LIN {X 0,Y 525.321,Z 367.806,A -85,B 0,C 180,E1 -4749.038,E2 -4749.038} C_VEL
LIN {X 0,Y 524.882,Z 392.684,A -85,B 0,C 180,E1 -4751.929,E2 -4751.929} C_VEL
LIN {X 0,Y 524.49,Z 417.897,A -85,B 0,C 180,E1 -4754.808,E2 -4754.808} C_VEL
LIN {X 0,Y 525.888,Z 431.517,A -85,B 0,C 180,E1 -4755.052,E2 -4755.052} C_VEL
LIN {X 0,Y 525.465,Z 528.308,A -85,B 0,C 180,E1 -4756.39,E2 -4756.39} C_VEL
LIN {X 0,Y 525.226,Z 541.664,A -85,B 0,C 180,E1 -4756.729,E2 -4756.729} C_VEL
LIN {X 0,Y 524.966,Z 553.932,A -85,B 0,C 180,E1 -4757.19,E2 -4757.19} C_VEL
LIN {X 0,Y 524.718,Z 566.459,A -85,B 0,C 180,E1 -4757.828,E2 -4757.828} C_VEL
LIN {X 0,Y 524.441,Z 578.107,A -85,B 0,C 180,E1 -4758.6,E2 -4758.6} C_VEL
LIN {X 0,Y 524.161,Z 588.71,A -85,B 0,C 180,E1 -4759.474,E2 -4759.474} C_VEL
LIN {X 0,Y 523.963,Z 597.402,A -85,B 0,C 180,E1 -4760.348,E2 -4760.348} C_VEL
LIN {X 0,Y 523.771,Z 605.435,A -85,B 0,C 180,E1 -4761.318,E2 -4761.318} C_VEL
LIN {X 0,Y 523.629,Z 613.302,A -85,B 0,C 180,E1 -4762.481,E2 -4762.481} C_VEL
LIN {X 0,Y 523.502,Z 620.559,A -85,B 0,C 180,E1 -4763.835,E2 -4763.835} C_VEL
LIN {X 0,Y 523.411,Z 625.392,A -85,B 0,C 180,E1 -4764.993,E2 -4764.993} C_VEL
LIN {X 0,Y 523.475,Z 629.106,A -85,B 0,C 180,E1 -4766.151,E2 -4766.151} C_VEL
LIN {X 0,Y 523.397,Z 631.008,A -85,B 0,C 180,E1 -4766.921,E2 -4766.921} C_VEL
LIN {X 0,Y 523.345,Z 632.435,A -85,B 0,C 180,E1 -4767.691,E2 -4767.691} C_VEL
LIN {X 0,Y 523.279,Z 634.074,A -85,B 0,C 180,E1 -4769.23,E2 -4769.23} C_VEL
LIN {X 0,Y 523.278,Z 634.296,A -85,B 0,C 180,E1 -4770,E2 -4770} C_VEL
LIN {X 0,Y 523.279,Z 634.074,A -85,B 0,C 180,E1 -4770.77,E2 -4770.77} C_VEL
LIN {X 0,Y 523.345,Z 632.438,A -85,B 0,C 180,E1 -4772.309,E2 -4772.309} C_VEL
LIN {X 0,Y 523.397,Z 631.011,A -85,B 0,C 180,E1 -4773.079,E2 -4773.079} C_VEL
LIN {X 0,Y 523.441,Z 628.004,A -85,B 0,C 180,E1 -4774.235,E2 -4774.235} C_VEL
LIN {X 0,Y 523.464,Z 623.93,A -85,B 0,C 180,E1 -4775.393,E2 -4775.393} C_VEL
LIN {X 0,Y 523.516,Z 618.58,A -85,B 0,C 180,E1 -4776.574,E2 -4776.574} C_VEL
LIN {X 0,Y 523.649,Z 612.112,A -85,B 0,C 180,E1 -4777.713,E2 -4777.713} C_VEL
LIN {X 0,Y 523.821,Z 603.92,A -85,B 0,C 180,E1 -4778.876,E2 -4778.876} C_VEL
LIN {X 0,Y 524.017,Z 595.588,A -85,B 0,C 180,E1 -4779.846,E2 -4779.846} C_VEL
LIN {X 0,Y 524.277,Z 585.449,A -85,B 0,C 180,E1 -4780.817,E2 -4780.817} C_VEL
LIN {X 0,Y 524.576,Z 573.997,A -85,B 0,C 180,E1 -4781.693,E2 -4781.693} C_VEL
LIN {X 0,Y 524.816,Z 562.855,A -85,B 0,C 180,E1 -4782.372,E2 -4782.372} C_VEL
LIN {X 0,Y 525.058,Z 550.507,A -85,B 0,C 180,E1 -4782.956,E2 -4782.956} C_VEL
LIN {X 0,Y 525.318,Z 537.59,A -85,B 0,C 180,E1 -4783.392,E2 -4783.392} C_VEL
LIN {X 0,Y 525.501,Z 523.939,A -85,B 0,C 180,E1 -4783.683,E2 -4783.683} C_VEL
LIN {X 0,Y 525.776,Z 428.93,A -85,B 0,C 180,E1 -4784.986,E2 -4784.986} C_VEL
LIN {X 0,Y 524.48,Z 417.737,A -85,B 0,C 180,E1 -4785.202,E2 -4785.202} C_VEL
LIN {X 0,Y 524.855,Z 393.85,A -85,B 0,C 180,E1 -4787.937,E2 -4787.937} C_VEL
LIN {X 0,Y 525.421,Z 366.009,A -85,B 0,C 180,E1 -4791.17,E2 -4791.17} C_VEL
LIN {X 0,Y 525.911,Z 339.704,A -85,B 0,C 180,E1 -4794.263,E2 -4794.263} C_VEL
LIN {X 0,Y 526.305,Z 318.022,A -85,B 0,C 180,E1 -4796.856,E2 -4796.856} C_VEL
LIN {X 0,Y 523.957,Z 306.361,A -85,B 0,C 180,E1 -4798.421,E2 -4798.421} C_VEL
LIN {X 0,Y 523.907,Z 306.224,A -85,B 0,C 180,E1 -4801.544,E2 -4801.544} C_VEL
LIN {X 0,Y 523.909,Z 306.226,A -85,B 0,C 180,E1 -4804.291,E2 -4804.291} C_VEL
LIN {X 0,Y 523.878,Z 306.229,A -85,B 0,C 180,E1 -4807.673,E2 -4807.673} C_VEL
LIN {X 0,Y 523.909,Z 306.223,A -85,B 0,C 180,E1 -4810.126,E2 -4810.126} C_VEL
LIN {X 0,Y 523.875,Z 306.224,A -85,B 0,C 180,E1 -4813.171,E2 -4813.171} C_VEL
LIN {X 0,Y 523.919,Z 306.214,A -85,B 0,C 180,E1 -4815.77,E2 -4815.77} C_VEL
LIN {X 0,Y 523.89,Z 306.223,A -85,B 0,C 180,E1 -4818.903,E2 -4818.903} C_VEL
LIN {X 0,Y 523.895,Z 306.213,A -85,B 0,C 180,E1 -4821.896,E2 -4821.896} C_VEL
LIN {X 0,Y 523.907,Z 306.212,A -85,B 0,C 180,E1 -4824.912,E2 -4824.912} C_VEL
LIN {X 0,Y 523.928,Z 306.222,A -85,B 0,C 180,E1 -4827.679,E2 -4827.679} C_VEL
LIN {X 0,Y 523.946,Z 306.211,A -85,B 0,C 180,E1 -4830.676,E2 -4830.676} C_VEL
LIN {X 0,Y 523.894,Z 306.226,A -85,B 0,C 180,E1 -4833.724,E2 -4833.724} C_VEL
LIN {X 0,Y 523.901,Z 306.222,A -85,B 0,C 180,E1 -4836.269,E2 -4836.269} C_VEL
LIN {X 0,Y 523.937,Z 306.208,A -85,B 0,C 180,E1 -4838.766,E2 -4838.766} C_VEL
LIN {X 0,Y 523.928,Z 306.214,A -85,B 0,C 180,E1 -4841.22,E2 -4841.22} C_VEL
LIN {X 0,Y 523.912,Z 306.226,A -85,B 0,C 180,E1 -4843.638,E2 -4843.638} C_VEL
LIN {X 0,Y 523.921,Z 306.219,A -85,B 0,C 180,E1 -4846.027,E2 -4846.027} C_VEL
LIN {X 0,Y 523.98,Z 306.211,A -85,B 0,C 180,E1 -4849.177,E2 -4849.177} C_VEL
LIN {X 0,Y 523.988,Z 306.209,A -85,B 0,C 180,E1 -4852.292,E2 -4852.292} C_VEL
LIN {X 0,Y 524.057,Z 306.198,A -85,B 0,C 180,E1 -4854.613,E2 -4854.613} C_VEL
LIN {X 0,Y 524.092,Z 306.206,A -85,B 0,C 180,E1 -4857.694,E2 -4857.694} C_VEL
LIN {X 0,Y 524.083,Z 306.197,A -85,B 0,C 180,E1 -4860,E2 -4860} C_VEL
LIN {X 0,Y 524.025,Z 306.205,A -85,B 0,C 180,E1 -4863.075,E2 -4863.075} C_VEL
LIN {X 0,Y 523.999,Z 306.208,A -85,B 0,C 180,E1 -4866.16,E2 -4866.16} C_VEL
LIN {X 0,Y 523.97,Z 306.212,A -85,B 0,C 180,E1 -4869.262,E2 -4869.262} C_VEL
LIN {X 0,Y 523.988,Z 306.216,A -85,B 0,C 180,E1 -4871.736,E2 -4871.736} C_VEL
LIN {X 0,Y 523.975,Z 306.208,A -85,B 0,C 180,E1 -4875.048,E2 -4875.048} C_VEL
LIN {X 0,Y 523.907,Z 306.223,A -85,B 0,C 180,E1 -4877.971,E2 -4877.971} C_VEL
LIN {X 0,Y 523.944,Z 306.212,A -85,B 0,C 180,E1 -4880.411,E2 -4880.411} C_VEL
LIN {X 0,Y 523.898,Z 306.221,A -85,B 0,C 180,E1 -4882.894,E2 -4882.894} C_VEL
LIN {X 0,Y 523.892,Z 306.229,A -85,B 0,C 180,E1 -4885.422,E2 -4885.422} C_VEL
LIN {X 0,Y 523.898,Z 306.213,A -85,B 0,C 180,E1 -4888.003,E2 -4888.003} C_VEL
LIN {X 0,Y 523.925,Z 306.208,A -85,B 0,C 180,E1 -4890.853,E2 -4890.853} C_VEL
LIN {X 0,Y 523.919,Z 306.224,A -85,B 0,C 180,E1 -4893.729,E2 -4893.729} C_VEL
LIN {X 0,Y 523.891,Z 306.22,A -85,B 0,C 180,E1 -4896.401,E2 -4896.401} C_VEL
LIN {X 0,Y 523.903,Z 306.216,A -85,B 0,C 180,E1 -4899.087,E2 -4899.087} C_VEL
LIN {X 0,Y 523.888,Z 306.223,A -85,B 0,C 180,E1 -4902.126,E2 -4902.126} C_VEL
LIN {X 0,Y 523.928,Z 306.223,A -85,B 0,C 180,E1 -4905.312,E2 -4905.312} C_VEL
LIN {X 0,Y 523.874,Z 306.219,A -85,B 0,C 180,E1 -4906.87,E2 -4906.87} C_VEL
LIN {X 0,Y 523.187,Z 306.312,A -85,B 0,C 180,E1 -4907.512,E2 -4907.512} C_VEL
LIN {X 0,Y 520.324,Z 306.668,A -85,B 0,C 180,E1 -4908.553,E2 -4908.553} C_VEL
LIN {X 0,Y 517.93,Z 306.972,A -85,B 0,C 180,E1 -4909.392,E2 -4909.392} C_VEL
LIN {X 0,Y 516.924,Z 307.092,A -85,B 0,C 180,E1 -4910.04,E2 -4910.04} C_VEL
LIN {X 0,Y 516.853,Z 307.099,A -85,B 0,C 180,E1 -4910.259,E2 -4910.259} C_VEL
LIN {X 0,Y 516.843,Z 307.102,A -85,B 0,C 180,E1 -4913.349,E2 -4913.349} C_VEL
LIN {X 0,Y 516.876,Z 307.096,A -85,B 0,C 180,E1 -4916.119,E2 -4916.119} C_VEL
LIN {X 0,Y 516.848,Z 307.102,A -85,B 0,C 180,E1 -4918.944,E2 -4918.944} C_VEL
LIN {X 0,Y 516.843,Z 307.094,A -85,B 0,C 180,E1 -4921.581,E2 -4921.581} C_VEL
LIN {X 0,Y 516.842,Z 307.1,A -85,B 0,C 180,E1 -4924.207,E2 -4924.207} C_VEL
LIN {X 0,Y 516.855,Z 307.102,A -85,B 0,C 180,E1 -4926.776,E2 -4926.776} C_VEL
LIN {X 0,Y 516.931,Z 307.093,A -85,B 0,C 180,E1 -4929.735,E2 -4929.735} C_VEL
LIN {X 0,Y 516.884,Z 307.07,A -85,B 0,C 180,E1 -4932.595,E2 -4932.595} C_VEL
LIN {X 0,Y 516.96,Z 307.275,A -85,B 0,C 180,E1 -4934.94,E2 -4934.94} C_VEL
LIN {X 0,Y 517.203,Z 308.319,A -85,B 0,C 180,E1 -4935.069,E2 -4935.069} C_VEL
LIN {X 0,Y 519.147,Z 313.948,A -85,B 0,C 180,E1 -4935.221,E2 -4935.221} C_VEL
LIN {X 0,Y 518.857,Z 387.345,A -85,B 0,C 180,E1 -4936.263,E2 -4936.263} C_VEL
LIN {X 0,Y 518.772,Z 400.457,A -85,B 0,C 180,E1 -4936.61,E2 -4936.61} C_VEL
LIN {X 0,Y 518.62,Z 413.364,A -85,B 0,C 180,E1 -4937.12,E2 -4937.12} C_VEL
LIN {X 0,Y 518.424,Z 425.059,A -85,B 0,C 180,E1 -4937.752,E2 -4937.752} C_VEL
LIN {X 0,Y 518.072,Z 436.629,A -85,B 0,C 180,E1 -4938.557,E2 -4938.557} C_VEL
LIN {X 0,Y 517.797,Z 446.757,A -85,B 0,C 180,E1 -4939.442,E2 -4939.442} C_VEL
LIN {X 0,Y 517.518,Z 455.832,A -85,B 0,C 180,E1 -4940.424,E2 -4940.424} C_VEL
LIN {X 0,Y 517.235,Z 464.615,A -85,B 0,C 180,E1 -4941.601,E2 -4941.601} C_VEL
LIN {X 0,Y 517.056,Z 470.802,A -85,B 0,C 180,E1 -4942.62,E2 -4942.62} C_VEL
LIN {X 0,Y 516.937,Z 476.425,A -85,B 0,C 180,E1 -4943.756,E2 -4943.756} C_VEL
LIN {X 0,Y 516.696,Z 481.059,A -85,B 0,C 180,E1 -4944.928,E2 -4944.928} C_VEL
LIN {X 0,Y 516.648,Z 484.586,A -85,B 0,C 180,E1 -4946.1,E2 -4946.1} C_VEL
LIN {X 0,Y 516.587,Z 486.413,A -85,B 0,C 180,E1 -4946.881,E2 -4946.881} C_VEL
LIN {X 0,Y 516.579,Z 487.788,A -85,B 0,C 180,E1 -4947.661,E2 -4947.661} C_VEL
LIN {X 0,Y 516.546,Z 489.367,A -85,B 0,C 180,E1 -4949.22,E2 -4949.22} C_VEL
LIN {X 0,Y 516.535,Z 489.601,A -85,B 0,C 180,E1 -4950,E2 -4950} C_VEL
LIN {X 0,Y 516.546,Z 489.421,A -85,B 0,C 180,E1 -4950.78,E2 -4950.78} C_VEL
LIN {X 0,Y 516.578,Z 487.91,A -85,B 0,C 180,E1 -4952.339,E2 -4952.339} C_VEL
LIN {X 0,Y 516.584,Z 486.591,A -85,B 0,C 180,E1 -4953.119,E2 -4953.119} C_VEL
LIN {X 0,Y 516.707,Z 483.784,A -85,B 0,C 180,E1 -4954.29,E2 -4954.29} C_VEL
LIN {X 0,Y 516.823,Z 479.981,A -85,B 0,C 180,E1 -4955.462,E2 -4955.462} C_VEL
LIN {X 0,Y 516.897,Z 474.869,A -85,B 0,C 180,E1 -4956.683,E2 -4956.683} C_VEL
LIN {X 0,Y 517.15,Z 467.686,A -85,B 0,C 180,E1 -4958.007,E2 -4958.007} C_VEL
LIN {X 0,Y 517.415,Z 459.672,A -85,B 0,C 180,E1 -4959.183,E2 -4959.183} C_VEL
LIN {X 0,Y 517.669,Z 451.454,A -85,B 0,C 180,E1 -4960.165,E2 -4960.165} C_VEL
LIN {X 0,Y 517.944,Z 442.436,A -85,B 0,C 180,E1 -4961.05,E2 -4961.05} C_VEL
LIN {X 0,Y 518.281,Z 431.958,A -85,B 0,C 180,E1 -4961.88,E2 -4961.88} C_VEL
LIN {X 0,Y 518.473,Z 420.319,A -85,B 0,C 180,E1 -4962.615,E2 -4962.615} C_VEL
LIN {X 0,Y 518.647,Z 408.922,A -85,B 0,C 180,E1 -4963.168,E2 -4963.168} C_VEL
LIN {X 0,Y 518.815,Z 396.128,A -85,B 0,C 180,E1 -4963.613,E2 -4963.613} C_VEL
LIN {X 0,Y 518.834,Z 383.996,A -85,B 0,C 180,E1 -4963.887,E2 -4963.887} C_VEL
LIN {X 0,Y 519.053,Z 313.676,A -85,B 0,C 180,E1 -4964.876,E2 -4964.876} C_VEL
LIN {X 0,Y 517.038,Z 307.902,A -85,B 0,C 180,E1 -4965.051,E2 -4965.051} C_VEL
LIN {X 0,Y 516.904,Z 307.157,A -85,B 0,C 180,E1 -4965.21,E2 -4965.21} C_VEL
LIN {X 0,Y 516.871,Z 307.068,A -85,B 0,C 180,E1 -4968.224,E2 -4968.224} C_VEL
LIN {X 0,Y 516.887,Z 307.104,A -85,B 0,C 180,E1 -4970.702,E2 -4970.702} C_VEL
LIN {X 0,Y 516.855,Z 307.102,A -85,B 0,C 180,E1 -4973.224,E2 -4973.224} C_VEL
LIN {X 0,Y 516.855,Z 307.099,A -85,B 0,C 180,E1 -4976.175,E2 -4976.175} C_VEL
LIN {X 0,Y 516.897,Z 307.095,A -85,B 0,C 180,E1 -4979.305,E2 -4979.305} C_VEL
LIN {X 0,Y 516.862,Z 307.101,A -85,B 0,C 180,E1 -4982.537,E2 -4982.537} C_VEL
LIN {X 0,Y 516.851,Z 307.1,A -85,B 0,C 180,E1 -4985.327,E2 -4985.327} C_VEL
LIN {X 0,Y 516.867,Z 307.102,A -85,B 0,C 180,E1 -4988.716,E2 -4988.716} C_VEL
LIN {X 0,Y 516.84,Z 307.098,A -85,B 0,C 180,E1 -4991.781,E2 -4991.781} C_VEL
LIN {X 0,Y 516.892,Z 307.098,A -85,B 0,C 180,E1 -4995.006,E2 -4995.006} C_VEL
LIN {X 0,Y 516.843,Z 307.106,A -85,B 0,C 180,E1 -4998.406,E2 -4998.406} C_VEL
LIN {X 0,Y 516.865,Z 307.089,A -85,B 0,C 180,E1 -5001.282,E2 -5001.282} C_VEL
LIN {X 0,Y 516.85,Z 307.101,A -85,B 0,C 180,E1 -5004.218,E2 -5004.218} C_VEL
LIN {X 0,Y 516.873,Z 307.096,A -85,B 0,C 180,E1 -5007.051,E2 -5007.051} C_VEL
LIN {X 0,Y 516.839,Z 307.089,A -85,B 0,C 180,E1 -5009.793,E2 -5009.793} C_VEL
LIN {X 0,Y 516.867,Z 307.094,A -85,B 0,C 180,E1 -5012.464,E2 -5012.464} C_VEL
LIN {X 0,Y 516.837,Z 307.103,A -85,B 0,C 180,E1 -5015.068,E2 -5015.068} C_VEL
LIN {X 0,Y 516.862,Z 307.096,A -85,B 0,C 180,E1 -5017.621,E2 -5017.621} C_VEL
LIN {X 0,Y 516.906,Z 307.092,A -85,B 0,C 180,E1 -5020.129,E2 -5020.129} C_VEL
LIN {X 0,Y 516.863,Z 307.096,A -85,B 0,C 180,E1 -5023.408,E2 -5023.408} C_VEL
LIN {X 0,Y 516.857,Z 307.094,A -85,B 0,C 180,E1 -5025.832,E2 -5025.832} C_VEL
LIN {X 0,Y 516.933,Z 307.09,A -85,B 0,C 180,E1 -5029.027,E2 -5029.027} C_VEL
LIN {X 0,Y 516.916,Z 307.093,A -85,B 0,C 180,E1 -5032.186,E2 -5032.186} C_VEL
LIN {X 0,Y 516.97,Z 307.091,A -85,B 0,C 180,E1 -5034.539,E2 -5034.539} C_VEL
LIN {X 0,Y 517.063,Z 307.072,A -85,B 0,C 180,E1 -5037.663,E2 -5037.663} C_VEL
LIN {X 0,Y 517.08,Z 307.072,A -85,B 0,C 180,E1 -5040.779,E2 -5040.779} C_VEL
LIN {X 0,Y 516.935,Z 307.088,A -85,B 0,C 180,E1 -5043.117,E2 -5043.117} C_VEL
LIN {X 0,Y 516.974,Z 307.086,A -85,B 0,C 180,E1 -5046.244,E2 -5046.244} C_VEL
LIN {X 0,Y 516.921,Z 307.09,A -85,B 0,C 180,E1 -5049.39,E2 -5049.39} C_VEL
LIN {X 0,Y 516.897,Z 307.094,A -85,B 0,C 180,E1 -5052.565,E2 -5052.565} C_VEL
LIN {X 0,Y 516.936,Z 307.088,A -85,B 0,C 180,E1 -5055.146,E2 -5055.146} C_VEL
LIN {X 0,Y 516.869,Z 307.101,A -85,B 0,C 180,E1 -5058.224,E2 -5058.224} C_VEL
LIN {X 0,Y 516.897,Z 307.088,A -85,B 0,C 180,E1 -5060.702,E2 -5060.702} C_VEL
LIN {X 0,Y 516.877,Z 307.102,A -85,B 0,C 180,E1 -5064.074,E2 -5064.074} C_VEL
LIN {X 0,Y 516.836,Z 307.1,A -85,B 0,C 180,E1 -5066.663,E2 -5066.663} C_VEL
LIN {X 0,Y 516.902,Z 307.09,A -85,B 0,C 180,E1 -5069.524,E2 -5069.524} C_VEL
LIN {X 0,Y 516.888,Z 307.097,A -85,B 0,C 180,E1 -5072.543,E2 -5072.543} C_VEL
LIN {X 0,Y 516.844,Z 307.097,A -85,B 0,C 180,E1 -5075.327,E2 -5075.327} C_VEL
LIN {X 0,Y 516.867,Z 307.095,A -85,B 0,C 180,E1 -5078.717,E2 -5078.717} C_VEL
LIN {X 0,Y 516.877,Z 307.101,A -85,B 0,C 180,E1 -5081.779,E2 -5081.779} C_VEL
LIN {X 0,Y 516.892,Z 307.082,A -85,B 0,C 180,E1 -5085.008,E2 -5085.008} C_VEL
LIN {X 0,Y 516.848,Z 307.102,A -85,B 0,C 180,E1 -5088.407,E2 -5088.407} C_VEL
LIN {X 0,Y 516.87,Z 307.095,A -85,B 0,C 180,E1 -5091.284,E2 -5091.284} C_VEL
LIN {X 0,Y 516.847,Z 307.101,A -85,B 0,C 180,E1 -5094.674,E2 -5094.674} C_VEL
LIN {X 0,Y 516.888,Z 307.094,A -85,B 0,C 180,E1 -5097.458,E2 -5097.458} C_VEL
LIN {X 0,Y 516.901,Z 307.077,A -85,B 0,C 180,E1 -5100.695,E2 -5100.695} C_VEL
LIN {X 0,Y 516.935,Z 307.345,A -85,B 0,C 180,E1 -5101.406,E2 -5101.406} C_VEL
LIN {X 0,Y 519.378,Z 319.028,A -85,B 0,C 180,E1 -5102.987,E2 -5102.987} C_VEL
LIN {X 0,Y 519.069,Z 337.058,A -85,B 0,C 180,E1 -5105.183,E2 -5105.183} C_VEL
LIN {X 0,Y 518.527,Z 361.62,A -85,B 0,C 180,E1 -5108.116,E2 -5108.116} C_VEL
LIN {X 0,Y 518.001,Z 386.005,A -85,B 0,C 180,E1 -5110.997,E2 -5110.997} C_VEL
LIN {X 0,Y 517.539,Z 410.213,A -85,B 0,C 180,E1 -5113.837,E2 -5113.837} C_VEL
LIN {X 0,Y 517.48,Z 416.952,A -85,B 0,C 180,E1 -5114.6,E2 -5114.6} C_VEL
LIN {X 0,Y 519.009,Z 432.102,A -85,B 0,C 180,E1 -5114.872,E2 -5114.872} C_VEL
LIN {X 0,Y 518.531,Z 527.315,A -85,B 0,C 180,E1 -5116.205,E2 -5116.205} C_VEL
LIN {X 0,Y 518.275,Z 540.67,A -85,B 0,C 180,E1 -5116.547,E2 -5116.547} C_VEL
LIN {X 0,Y 518.014,Z 552.939,A -85,B 0,C 180,E1 -5117.015,E2 -5117.015} C_VEL
LIN {X 0,Y 517.708,Z 565.493,A -85,B 0,C 180,E1 -5117.663,E2 -5117.663} C_VEL
LIN {X 0,Y 517.439,Z 577.113,A -85,B 0,C 180,E1 -5118.443,E2 -5118.443} C_VEL
LIN {X 0,Y 517.134,Z 587.715,A -85,B 0,C 180,E1 -5119.329,E2 -5119.329} C_VEL
LIN {X 0,Y 516.911,Z 596.406,A -85,B 0,C 180,E1 -5120.215,E2 -5120.215} C_VEL
LIN {X 0,Y 516.711,Z 604.441,A -85,B 0,C 180,E1 -5121.198,E2 -5121.198} C_VEL
LIN {X 0,Y 516.554,Z 612.309,A -85,B 0,C 180,E1 -5122.377,E2 -5122.377} C_VEL
LIN {X 0,Y 516.435,Z 619.57,A -85,B 0,C 180,E1 -5123.75,E2 -5123.75} C_VEL
LIN {X 0,Y 516.382,Z 624.41,A -85,B 0,C 180,E1 -5124.925,E2 -5124.925} C_VEL
LIN {X 0,Y 516.43,Z 628.124,A -85,B 0,C 180,E1 -5126.098,E2 -5126.098} C_VEL
LIN {X 0,Y 516.352,Z 630.026,A -85,B 0,C 180,E1 -5126.879,E2 -5126.879} C_VEL
LIN {X 0,Y 516.304,Z 631.455,A -85,B 0,C 180,E1 -5127.66,E2 -5127.66} C_VEL
LIN {X 0,Y 516.265,Z 633.098,A -85,B 0,C 180,E1 -5129.22,E2 -5129.22} C_VEL
LIN {X 0,Y 516.261,Z 633.319,A -85,B 0,C 180,E1 -5130,E2 -5130} C_VEL
LIN {X 0,Y 516.265,Z 633.098,A -85,B 0,C 180,E1 -5130.78,E2 -5130.78} C_VEL
LIN {X 0,Y 516.304,Z 631.458,A -85,B 0,C 180,E1 -5132.34,E2 -5132.34} C_VEL
LIN {X 0,Y 516.352,Z 630.029,A -85,B 0,C 180,E1 -5133.121,E2 -5133.121} C_VEL
LIN {X 0,Y 516.387,Z 627.02,A -85,B 0,C 180,E1 -5134.293,E2 -5134.293} C_VEL
LIN {X 0,Y 516.404,Z 622.943,A -85,B 0,C 180,E1 -5135.467,E2 -5135.467} C_VEL
LIN {X 0,Y 516.489,Z 616.818,A -85,B 0,C 180,E1 -5136.812,E2 -5136.812} C_VEL
LIN {X 0,Y 516.585,Z 609.855,A -85,B 0,C 180,E1 -5138.016,E2 -5138.016} C_VEL
LIN {X 0,Y 516.769,Z 601.403,A -85,B 0,C 180,E1 -5139.195,E2 -5139.195} C_VEL
LIN {X 0,Y 517.006,Z 592.757,A -85,B 0,C 180,E1 -5140.178,E2 -5140.178} C_VEL
LIN {X 0,Y 517.318,Z 582.101,A -85,B 0,C 180,E1 -5141.162,E2 -5141.162} C_VEL
LIN {X 0,Y 517.578,Z 571.208,A -85,B 0,C 180,E1 -5141.976,E2 -5141.976} C_VEL
LIN {X 0,Y 517.86,Z 560.07,A -85,B 0,C 180,E1 -5142.64,E2 -5142.64} C_VEL
LIN {X 0,Y 518.18,Z 548.294,A -85,B 0,C 180,E1 -5143.181,E2 -5143.181} C_VEL
LIN {X 0,Y 518.403,Z 535.678,A -85,B 0,C 180,E1 -5143.599,E2 -5143.599} C_VEL
LIN {X 0,Y 518.601,Z 522.951,A -85,B 0,C 180,E1 -5143.868,E2 -5143.868} C_VEL
LIN {X 0,Y 518.903,Z 429.886,A -85,B 0,C 180,E1 -5145.162,E2 -5145.162} C_VEL
LIN {X 0,Y 517.455,Z 416.853,A -85,B 0,C 180,E1 -5145.406,E2 -5145.406} C_VEL
LIN {X 0,Y 517.899,Z 391.373,A -85,B 0,C 180,E1 -5148.37,E2 -5148.37} C_VEL
LIN {X 0,Y 518.44,Z 365.117,A -85,B 0,C 180,E1 -5151.47,E2 -5151.47} C_VEL
LIN {X 0,Y 518.976,Z 340.569,A -85,B 0,C 180,E1 -5154.395,E2 -5154.395} C_VEL
LIN {X 0,Y 519.465,Z 320.55,A -85,B 0,C 180,E1 -5156.819,E2 -5156.819} C_VEL
LIN {X 0,Y 518.03,Z 312.209,A -85,B 0,C 180,E1 -5157.917,E2 -5157.917} C_VEL
LIN {X 0,Y 516.899,Z 307.213,A -85,B 0,C 180,E1 -5158.638,E2 -5158.638} C_VEL
LIN {X 0,Y 516.877,Z 307.098,A -85,B 0,C 180,E1 -5161.11,E2 -5161.11} C_VEL
LIN {X 0,Y 516.879,Z 307.103,A -85,B 0,C 180,E1 -5163.961,E2 -5163.961} C_VEL
LIN {X 0,Y 516.812,Z 307.106,A -85,B 0,C 180,E1 -5166.751,E2 -5166.751} C_VEL
LIN {X 0,Y 516.854,Z 307.098,A -85,B 0,C 180,E1 -5169.723,E2 -5169.723} C_VEL
LIN {X 0,Y 516.837,Z 307.101,A -85,B 0,C 180,E1 -5172.835,E2 -5172.835} C_VEL
LIN {X 0,Y 516.891,Z 307.083,A -85,B 0,C 180,E1 -5175.006,E2 -5175.006} C_VEL
LIN {X 0,Y 516.88,Z 307.099,A -85,B 0,C 180,E1 -5178.402,E2 -5178.402} C_VEL
LIN {X 0,Y 516.867,Z 307.093,A -85,B 0,C 180,E1 -5181.283,E2 -5181.283} C_VEL
LIN {X 0,Y 516.844,Z 307.092,A -85,B 0,C 180,E1 -5184.672,E2 -5184.672} C_VEL
LIN {X 0,Y 516.887,Z 307.096,A -85,B 0,C 180,E1 -5187.457,E2 -5187.457} C_VEL
LIN {X 0,Y 516.914,Z 307.086,A -85,B 0,C 180,E1 -5190.695,E2 -5190.695} C_VEL
LIN {X 0,Y 516.873,Z 307.102,A -85,B 0,C 180,E1 -5193.818,E2 -5193.818} C_VEL
LIN {X 0,Y 516.85,Z 307.097,A -85,B 0,C 180,E1 -5196.775,E2 -5196.775} C_VEL
LIN {X 0,Y 516.929,Z 307.087,A -85,B 0,C 180,E1 -5199.732,E2 -5199.732} C_VEL
LIN {X 0,Y 516.886,Z 307.094,A -85,B 0,C 180,E1 -5202.595,E2 -5202.595} C_VEL
LIN {X 0,Y 516.934,Z 307.089,A -85,B 0,C 180,E1 -5205.03,E2 -5205.03} C_VEL
LIN {X 0,Y 516.958,Z 307.087,A -85,B 0,C 180,E1 -5208.233,E2 -5208.233} C_VEL
LIN {X 0,Y 516.92,Z 307.094,A -85,B 0,C 180,E1 -5211.399,E2 -5211.399} C_VEL
LIN {X 0,Y 516.976,Z 307.086,A -85,B 0,C 180,E1 -5213.756,E2 -5213.756} C_VEL
LIN {X 0,Y 516.937,Z 307.088,A -85,B 0,C 180,E1 -5216.883,E2 -5216.883} C_VEL
LIN {X 0,Y 517.08,Z 307.072,A -85,B 0,C 180,E1 -5219.221,E2 -5219.221} C_VEL
LIN {X 0,Y 517.064,Z 307.072,A -85,B 0,C 180,E1 -5222.337,E2 -5222.337} C_VEL
LIN {X 0,Y 516.964,Z 307.083,A -85,B 0,C 180,E1 -5226.244,E2 -5226.244} C_VEL
LIN {X 0,Y 516.927,Z 307.091,A -85,B 0,C 180,E1 -5229.39,E2 -5229.39} C_VEL
LIN {X 0,Y 516.944,Z 307.092,A -85,B 0,C 180,E1 -5231.807,E2 -5231.807} C_VEL
LIN {X 0,Y 516.928,Z 307.086,A -85,B 0,C 180,E1 -5235.143,E2 -5235.143} C_VEL
LIN {X 0,Y 516.869,Z 307.097,A -85,B 0,C 180,E1 -5238.224,E2 -5238.224} C_VEL
LIN {X 0,Y 516.894,Z 307.09,A -85,B 0,C 180,E1 -5240.702,E2 -5240.702} C_VEL
LIN {X 0,Y 516.848,Z 307.103,A -85,B 0,C 180,E1 -5243.225,E2 -5243.225} C_VEL
LIN {X 0,Y 516.873,Z 307.094,A -85,B 0,C 180,E1 -5246.182,E2 -5246.182} C_VEL
LIN {X 0,Y 516.896,Z 307.085,A -85,B 0,C 180,E1 -5249.306,E2 -5249.306} C_VEL
LIN {X 0,Y 516.887,Z 307.091,A -85,B 0,C 180,E1 -5252.543,E2 -5252.543} C_VEL
LIN {X 0,Y 516.854,Z 307.106,A -85,B 0,C 180,E1 -5255.329,E2 -5255.329} C_VEL
LIN {X 0,Y 516.87,Z 307.09,A -85,B 0,C 180,E1 -5257.943,E2 -5257.943} C_VEL
LIN {X 0,Y 516.842,Z 307.095,A -85,B 0,C 180,E1 -5260.746,E2 -5260.746} C_VEL
LIN {X 0,Y 516.876,Z 307.098,A -85,B 0,C 180,E1 -5263.904,E2 -5263.904} C_VEL
LIN {X 0,Y 516.825,Z 307.097,A -85,B 0,C 180,E1 -5266.872,E2 -5266.872} C_VEL
LIN {X 0,Y 516.855,Z 307.105,A -85,B 0,C 180,E1 -5269.594,E2 -5269.594} C_VEL
LIN {X 0,Y 516.853,Z 307.099,A -85,B 0,C 180,E1 -5270.259,E2 -5270.259} C_VEL
LIN {X 0,Y 516.215,Z 307.182,A -85,B 0,C 180,E1 -5270.909,E2 -5270.909} C_VEL
LIN {X 0,Y 513.368,Z 307.541,A -85,B 0,C 180,E1 -5271.965,E2 -5271.965} C_VEL
LIN {X 0,Y 510.938,Z 307.845,A -85,B 0,C 180,E1 -5272.815,E2 -5272.815} C_VEL
LIN {X 0,Y 509.887,Z 307.973,A -85,B 0,C 180,E1 -5273.471,E2 -5273.471} C_VEL
LIN {X 0,Y 509.799,Z 307.982,A -85,B 0,C 180,E1 -5273.694,E2 -5273.694} C_VEL
LIN {X 0,Y 509.831,Z 307.973,A -85,B 0,C 180,E1 -5276.538,E2 -5276.538} C_VEL
LIN {X 0,Y 509.804,Z 307.986,A -85,B 0,C 180,E1 -5279.332,E2 -5279.332} C_VEL
LIN {X 0,Y 509.826,Z 307.963,A -85,B 0,C 180,E1 -5282.051,E2 -5282.051} C_VEL
LIN {X 0,Y 509.783,Z 307.981,A -85,B 0,C 180,E1 -5284.699,E2 -5284.699} C_VEL
LIN {X 0,Y 509.825,Z 307.972,A -85,B 0,C 180,E1 -5287.459,E2 -5287.459} C_VEL
LIN {X 0,Y 509.907,Z 307.967,A -85,B 0,C 180,E1 -5289.845,E2 -5289.845} C_VEL
LIN {X 0,Y 509.82,Z 307.947,A -85,B 0,C 180,E1 -5293.173,E2 -5293.173} C_VEL
LIN {X 0,Y 509.902,Z 308.111,A -85,B 0,C 180,E1 -5294.711,E2 -5294.711} C_VEL
LIN {X 0,Y 510.083,Z 308.927,A -85,B 0,C 180,E1 -5294.84,E2 -5294.84} C_VEL
LIN {X 0,Y 512.276,Z 315.271,A -85,B 0,C 180,E1 -5295.022,E2 -5295.022} C_VEL
LIN {X 0,Y 512.032,Z 388.351,A -85,B 0,C 180,E1 -5296.077,E2 -5296.077} C_VEL
LIN {X 0,Y 511.929,Z 401.454,A -85,B 0,C 180,E1 -5296.428,E2 -5296.428} C_VEL
LIN {X 0,Y 511.766,Z 414.356,A -85,B 0,C 180,E1 -5296.944,E2 -5296.944} C_VEL
LIN {X 0,Y 511.589,Z 425.155,A -85,B 0,C 180,E1 -5297.529,E2 -5297.529} C_VEL
LIN {X 0,Y 511.227,Z 436.344,A -85,B 0,C 180,E1 -5298.301,E2 -5298.301} C_VEL
LIN {X 0,Y 510.917,Z 446.693,A -85,B 0,C 180,E1 -5299.198,E2 -5299.198} C_VEL
LIN {X 0,Y 510.663,Z 455.133,A -85,B 0,C 180,E1 -5300.094,E2 -5300.094} C_VEL
LIN {X 0,Y 510.345,Z 462.903,A -85,B 0,C 180,E1 -5301.088,E2 -5301.088} C_VEL
LIN {X 0,Y 510.122,Z 470.588,A -85,B 0,C 180,E1 -5302.3,E2 -5302.3} C_VEL
LIN {X 0,Y 509.954,Z 477.406,A -85,B 0,C 180,E1 -5303.67,E2 -5303.67} C_VEL
LIN {X 0,Y 509.699,Z 482.038,A -85,B 0,C 180,E1 -5304.858,E2 -5304.858} C_VEL
LIN {X 0,Y 509.633,Z 485.566,A -85,B 0,C 180,E1 -5306.046,E2 -5306.046} C_VEL
LIN {X 0,Y 509.565,Z 487.393,A -85,B 0,C 180,E1 -5306.838,E2 -5306.838} C_VEL
LIN {X 0,Y 509.568,Z 488.765,A -85,B 0,C 180,E1 -5307.629,E2 -5307.629} C_VEL
LIN {X 0,Y 509.533,Z 490.343,A -85,B 0,C 180,E1 -5309.21,E2 -5309.21} C_VEL
LIN {X 0,Y 509.521,Z 490.577,A -85,B 0,C 180,E1 -5310,E2 -5310} C_VEL
LIN {X 0,Y 509.533,Z 490.396,A -85,B 0,C 180,E1 -5310.79,E2 -5310.79} C_VEL
LIN {X 0,Y 509.568,Z 488.885,A -85,B 0,C 180,E1 -5312.371,E2 -5312.371} C_VEL
LIN {X 0,Y 509.562,Z 487.568,A -85,B 0,C 180,E1 -5313.163,E2 -5313.163} C_VEL
LIN {X 0,Y 509.695,Z 484.761,A -85,B 0,C 180,E1 -5314.349,E2 -5314.349} C_VEL
LIN {X 0,Y 509.84,Z 480.956,A -85,B 0,C 180,E1 -5315.537,E2 -5315.537} C_VEL
LIN {X 0,Y 509.916,Z 475.854,A -85,B 0,C 180,E1 -5316.773,E2 -5316.773} C_VEL
LIN {X 0,Y 510.194,Z 468.66,A -85,B 0,C 180,E1 -5318.117,E2 -5318.117} C_VEL
LIN {X 0,Y 510.484,Z 460.644,A -85,B 0,C 180,E1 -5319.309,E2 -5319.309} C_VEL
LIN {X 0,Y 510.753,Z 452.426,A -85,B 0,C 180,E1 -5320.304,E2 -5320.304} C_VEL
LIN {X 0,Y 511.046,Z 443.407,A -85,B 0,C 180,E1 -5321.201,E2 -5321.201} C_VEL
LIN {X 0,Y 511.412,Z 432.926,A -85,B 0,C 180,E1 -5322.042,E2 -5322.042} C_VEL
LIN {X 0,Y 511.617,Z 421.286,A -85,B 0,C 180,E1 -5322.787,E2 -5322.787} C_VEL
LIN {X 0,Y 511.795,Z 409.887,A -85,B 0,C 180,E1 -5323.348,E2 -5323.348} C_VEL
LIN {X 0,Y 511.971,Z 397.086,A -85,B 0,C 180,E1 -5323.799,E2 -5323.799} C_VEL
LIN {X 0,Y 511.993,Z 384.94,A -85,B 0,C 180,E1 -5324.076,E2 -5324.076} C_VEL
LIN {X 0,Y 512.276,Z 315.283,A -85,B 0,C 180,E1 -5325.068,E2 -5325.068} C_VEL
LIN {X 0,Y 510.03,Z 308.901,A -85,B 0,C 180,E1 -5325.254,E2 -5325.254} C_VEL
LIN {X 0,Y 509.838,Z 308.05,A -85,B 0,C 180,E1 -5325.415,E2 -5325.415} C_VEL
LIN {X 0,Y 509.828,Z 307.949,A -85,B 0,C 180,E1 -5328.485,E2 -5328.485} C_VEL
LIN {X 0,Y 509.834,Z 307.977,A -85,B 0,C 180,E1 -5331.002,E2 -5331.002} C_VEL
LIN {X 0,Y 509.811,Z 307.977,A -85,B 0,C 180,E1 -5333.564,E2 -5333.564} C_VEL
LIN {X 0,Y 509.796,Z 307.978,A -85,B 0,C 180,E1 -5336.351,E2 -5336.351} C_VEL
LIN {X 0,Y 509.83,Z 307.973,A -85,B 0,C 180,E1 -5338.847,E2 -5338.847} C_VEL
LIN {X 0,Y 509.786,Z 307.979,A -85,B 0,C 180,E1 -5341.592,E2 -5341.592} C_VEL
LIN {X 0,Y 509.827,Z 307.978,A -85,B 0,C 180,E1 -5344.415,E2 -5344.415} C_VEL
LIN {X 0,Y 509.789,Z 307.975,A -85,B 0,C 180,E1 -5347.342,E2 -5347.342} C_VEL
LIN {X 0,Y 509.809,Z 307.981,A -85,B 0,C 180,E1 -5350.384,E2 -5350.384} C_VEL
LIN {X 0,Y 509.788,Z 307.971,A -85,B 0,C 180,E1 -5353.574,E2 -5353.574} C_VEL
LIN {X 0,Y 509.786,Z 307.985,A -85,B 0,C 180,E1 -5356.424,E2 -5356.424} C_VEL
LIN {X 0,Y 509.807,Z 307.97,A -85,B 0,C 180,E1 -5359.614,E2 -5359.614} C_VEL
LIN {X 0,Y 509.798,Z 307.979,A -85,B 0,C 180,E1 -5362.657,E2 -5362.657} C_VEL
LIN {X 0,Y 509.832,Z 307.974,A -85,B 0,C 180,E1 -5365.8,E2 -5365.8} C_VEL
LIN {X 0,Y 509.831,Z 307.967,A -85,B 0,C 180,E1 -5368.721,E2 -5368.721} C_VEL
LIN {X 0,Y 509.808,Z 307.965,A -85,B 0,C 180,E1 -5371.916,E2 -5371.916} C_VEL
LIN {X 0,Y 509.794,Z 307.984,A -85,B 0,C 180,E1 -5374.699,E2 -5374.699} C_VEL
LIN {X 0,Y 509.816,Z 307.974,A -85,B 0,C 180,E1 -5377.459,E2 -5377.459} C_VEL
LIN {X 0,Y 509.881,Z 307.964,A -85,B 0,C 180,E1 -5379.843,E2 -5379.843} C_VEL
LIN {X 0,Y 509.81,Z 307.976,A -85,B 0,C 180,E1 -5383.172,E2 -5383.172} C_VEL
LIN {X 0,Y 509.832,Z 307.967,A -85,B 0,C 180,E1 -5385.633,E2 -5385.633} C_VEL
LIN {X 0,Y 509.898,Z 307.968,A -85,B 0,C 180,E1 -5388.874,E2 -5388.874} C_VEL
LIN {X 0,Y 509.868,Z 307.969,A -85,B 0,C 180,E1 -5392.077,E2 -5392.077} C_VEL
LIN {X 0,Y 509.923,Z 307.97,A -85,B 0,C 180,E1 -5394.464,E2 -5394.464} C_VEL
LIN {X 0,Y 510.034,Z 307.947,A -85,B 0,C 180,E1 -5397.631,E2 -5397.631} C_VEL
LIN {X 0,Y 510.029,Z 307.95,A -85,B 0,C 180,E1 -5400.79,E2 -5400.79} C_VEL
LIN {X 0,Y 509.879,Z 307.967,A -85,B 0,C 180,E1 -5403.161,E2 -5403.161} C_VEL
LIN {X 0,Y 509.928,Z 307.963,A -85,B 0,C 180,E1 -5406.33,E2 -5406.33} C_VEL
LIN {X 0,Y 509.873,Z 307.971,A -85,B 0,C 180,E1 -5408.721,E2 -5408.721} C_VEL
LIN {X 0,Y 509.892,Z 307.968,A -85,B 0,C 180,E1 -5411.932,E2 -5411.932} C_VEL
LIN {X 0,Y 509.887,Z 307.966,A -85,B 0,C 180,E1 -5415.242,E2 -5415.242} C_VEL
LIN {X 0,Y 509.829,Z 307.973,A -85,B 0,C 180,E1 -5418.485,E2 -5418.485} C_VEL
LIN {X 0,Y 509.838,Z 307.964,A -85,B 0,C 180,E1 -5421.002,E2 -5421.002} C_VEL
LIN {X 0,Y 509.811,Z 307.976,A -85,B 0,C 180,E1 -5423.564,E2 -5423.564} C_VEL
LIN {X 0,Y 509.81,Z 307.979,A -85,B 0,C 180,E1 -5426.357,E2 -5426.357} C_VEL
LIN {X 0,Y 509.842,Z 307.968,A -85,B 0,C 180,E1 -5428.846,E2 -5428.846} C_VEL
LIN {X 0,Y 509.812,Z 307.978,A -85,B 0,C 180,E1 -5431.591,E2 -5431.591} C_VEL
LIN {X 0,Y 509.827,Z 307.975,A -85,B 0,C 180,E1 -5434.415,E2 -5434.415} C_VEL
LIN {X 0,Y 509.774,Z 307.982,A -85,B 0,C 180,E1 -5437.345,E2 -5437.345} C_VEL
LIN {X 0,Y 509.808,Z 307.981,A -85,B 0,C 180,E1 -5440.385,E2 -5440.385} C_VEL
LIN {X 0,Y 509.79,Z 307.976,A -85,B 0,C 180,E1 -5443.059,E2 -5443.059} C_VEL
LIN {X 0,Y 509.802,Z 307.97,A -85,B 0,C 180,E1 -5445.796,E2 -5445.796} C_VEL
LIN {X 0,Y 509.801,Z 307.978,A -85,B 0,C 180,E1 -5448.57,E2 -5448.57} C_VEL
LIN {X 0,Y 509.812,Z 307.977,A -85,B 0,C 180,E1 -5451.659,E2 -5451.659} C_VEL
LIN {X 0,Y 509.805,Z 307.978,A -85,B 0,C 180,E1 -5454.621,E2 -5454.621} C_VEL
LIN {X 0,Y 509.854,Z 307.971,A -85,B 0,C 180,E1 -5457.481,E2 -5457.481} C_VEL
LIN {X 0,Y 509.865,Z 307.953,A -85,B 0,C 180,E1 -5460.93,E2 -5460.93} C_VEL
LIN {X 0,Y 509.878,Z 308.244,A -85,B 0,C 180,E1 -5461.203,E2 -5461.203} C_VEL
LIN {X 0,Y 512.493,Z 320.566,A -85,B 0,C 180,E1 -5462.895,E2 -5462.895} C_VEL
LIN {X 0,Y 512.063,Z 341.516,A -85,B 0,C 180,E1 -5465.479,E2 -5465.479} C_VEL
LIN {X 0,Y 511.4,Z 367.717,A -85,B 0,C 180,E1 -5468.643,E2 -5468.643} C_VEL
LIN {X 0,Y 510.833,Z 393.06,A -85,B 0,C 180,E1 -5471.677,E2 -5471.677} C_VEL
LIN {X 0,Y 510.451,Z 415.836,A -85,B 0,C 180,E1 -5474.375,E2 -5474.375} C_VEL
LIN {X 0,Y 512.128,Z 433.473,A -85,B 0,C 180,E1 -5474.697,E2 -5474.697} C_VEL
LIN {X 0,Y 511.635,Z 526.326,A -85,B 0,C 180,E1 -5476.015,E2 -5476.015} C_VEL
LIN {X 0,Y 511.371,Z 539.682,A -85,B 0,C 180,E1 -5476.362,E2 -5476.362} C_VEL
LIN {X 0,Y 511.023,Z 553.079,A -85,B 0,C 180,E1 -5476.884,E2 -5476.884} C_VEL
LIN {X 0,Y 510.683,Z 565.385,A -85,B 0,C 180,E1 -5477.547,E2 -5477.547} C_VEL
LIN {X 0,Y 510.386,Z 577.427,A -85,B 0,C 180,E1 -5478.382,E2 -5478.382} C_VEL
LIN {X 0,Y 510.065,Z 587.784,A -85,B 0,C 180,E1 -5479.28,E2 -5479.28} C_VEL
LIN {X 0,Y 509.792,Z 597.123,A -85,B 0,C 180,E1 -5480.278,E2 -5480.278} C_VEL
LIN {X 0,Y 509.594,Z 606.246,A -85,B 0,C 180,E1 -5481.474,E2 -5481.474} C_VEL
LIN {X 0,Y 509.436,Z 613.603,A -85,B 0,C 180,E1 -5482.669,E2 -5482.669} C_VEL
LIN {X 0,Y 509.367,Z 618.58,A -85,B 0,C 180,E1 -5483.663,E2 -5483.663} C_VEL
LIN {X 0,Y 509.33,Z 623.425,A -85,B 0,C 180,E1 -5484.854,E2 -5484.854} C_VEL
LIN {X 0,Y 509.385,Z 627.141,A -85,B 0,C 180,E1 -5486.044,E2 -5486.044} C_VEL
LIN {X 0,Y 509.306,Z 629.044,A -85,B 0,C 180,E1 -5486.836,E2 -5486.836} C_VEL
LIN {X 0,Y 509.263,Z 630.474,A -85,B 0,C 180,E1 -5487.627,E2 -5487.627} C_VEL
LIN {X 0,Y 509.25,Z 632.121,A -85,B 0,C 180,E1 -5489.209,E2 -5489.209} C_VEL
LIN {X 0,Y 509.244,Z 632.343,A -85,B 0,C 180,E1 -5490,E2 -5490} C_VEL
LIN {X 0,Y 509.25,Z 632.122,A -85,B 0,C 180,E1 -5490.791,E2 -5490.791} C_VEL
LIN {X 0,Y 509.263,Z 630.477,A -85,B 0,C 180,E1 -5492.373,E2 -5492.373} C_VEL
LIN {X 0,Y 509.306,Z 629.048,A -85,B 0,C 180,E1 -5493.164,E2 -5493.164} C_VEL
LIN {X 0,Y 509.337,Z 626.036,A -85,B 0,C 180,E1 -5494.352,E2 -5494.352} C_VEL
LIN {X 0,Y 509.344,Z 621.956,A -85,B 0,C 180,E1 -5495.543,E2 -5495.543} C_VEL
LIN {X 0,Y 509.417,Z 616.053,A -85,B 0,C 180,E1 -5496.864,E2 -5496.864} C_VEL
LIN {X 0,Y 509.535,Z 608.864,A -85,B 0,C 180,E1 -5498.127,E2 -5498.127} C_VEL
LIN {X 0,Y 509.71,Z 600.408,A -85,B 0,C 180,E1 -5499.324,E2 -5499.324} C_VEL
LIN {X 0,Y 509.953,Z 591.759,A -85,B 0,C 180,E1 -5500.321,E2 -5500.321} C_VEL
LIN {X 0,Y 510.217,Z 581.094,A -85,B 0,C 180,E1 -5501.32,E2 -5501.32} C_VEL
LIN {X 0,Y 510.535,Z 570.206,A -85,B 0,C 180,E1 -5502.144,E2 -5502.144} C_VEL
LIN {X 0,Y 510.839,Z 559.068,A -85,B 0,C 180,E1 -5502.817,E2 -5502.817} C_VEL
LIN {X 0,Y 511.245,Z 547.302,A -85,B 0,C 180,E1 -5503.363,E2 -5503.363} C_VEL
LIN {X 0,Y 511.458,Z 534.684,A -85,B 0,C 180,E1 -5503.787,E2 -5503.787} C_VEL
LIN {X 0,Y 511.716,Z 521.963,A -85,B 0,C 180,E1 -5504.059,E2 -5504.059} C_VEL
LIN {X 0,Y 511.975,Z 429.992,A -85,B 0,C 180,E1 -5505.357,E2 -5505.357} C_VEL
LIN {X 0,Y 510.429,Z 415.856,A -85,B 0,C 180,E1 -5505.625,E2 -5505.625} C_VEL
LIN {X 0,Y 510.895,Z 390.289,A -85,B 0,C 180,E1 -5508.652,E2 -5508.652} C_VEL
LIN {X 0,Y 511.459,Z 365.977,A -85,B 0,C 180,E1 -5511.566,E2 -5511.566} C_VEL
LIN {X 0,Y 512.049,Z 341.515,A -85,B 0,C 180,E1 -5514.521,E2 -5514.521} C_VEL
LIN {X 0,Y 512.558,Z 321.608,A -85,B 0,C 180,E1 -5516.968,E2 -5516.968} C_VEL
LIN {X 0,Y 510.713,Z 311.946,A -85,B 0,C 180,E1 -5518.271,E2 -5518.271} C_VEL
LIN {X 0,Y 509.858,Z 308.086,A -85,B 0,C 180,E1 -5518.845,E2 -5518.845} C_VEL
LIN {X 0,Y 509.81,Z 307.981,A -85,B 0,C 180,E1 -5521.59,E2 -5521.59} C_VEL
LIN {X 0,Y 509.831,Z 307.978,A -85,B 0,C 180,E1 -5524.414,E2 -5524.414} C_VEL
LIN {X 0,Y 509.78,Z 307.982,A -85,B 0,C 180,E1 -5527.343,E2 -5527.343} C_VEL
LIN {X 0,Y 509.809,Z 307.98,A -85,B 0,C 180,E1 -5530.384,E2 -5530.384} C_VEL
LIN {X 0,Y 509.801,Z 307.981,A -85,B 0,C 180,E1 -5533.573,E2 -5533.573} C_VEL
LIN {X 0,Y 509.803,Z 307.978,A -85,B 0,C 180,E1 -5536.426,E2 -5536.426} C_VEL
LIN {X 0,Y 509.806,Z 307.979,A -85,B 0,C 180,E1 -5539.305,E2 -5539.305} C_VEL
LIN {X 0,Y 509.808,Z 307.967,A -85,B 0,C 180,E1 -5541.791,E2 -5541.791} C_VEL
LIN {X 0,Y 509.806,Z 307.969,A -85,B 0,C 180,E1 -5544.62,E2 -5544.62} C_VEL
LIN {X 0,Y 509.853,Z 307.973,A -85,B 0,C 180,E1 -5547.48,E2 -5547.48} C_VEL
LIN {X 0,Y 509.852,Z 307.969,A -85,B 0,C 180,E1 -5550.273,E2 -5550.273} C_VEL
LIN {X 0,Y 509.823,Z 307.971,A -85,B 0,C 180,E1 -5552.941,E2 -5552.941} C_VEL
LIN {X 0,Y 509.827,Z 307.979,A -85,B 0,C 180,E1 -5555.572,E2 -5555.572} C_VEL
LIN {X 0,Y 509.813,Z 307.971,A -85,B 0,C 180,E1 -5558.148,E2 -5558.148} C_VEL
LIN {X 0,Y 509.847,Z 307.966,A -85,B 0,C 180,E1 -5560.681,E2 -5560.681} C_VEL
LIN {X 0,Y 509.855,Z 307.971,A -85,B 0,C 180,E1 -5563.174,E2 -5563.174} C_VEL
LIN {X 0,Y 509.85,Z 307.978,A -85,B 0,C 180,E1 -5565.634,E2 -5565.634} C_VEL
LIN {X 0,Y 509.901,Z 307.963,A -85,B 0,C 180,E1 -5568.874,E2 -5568.874} C_VEL
LIN {X 0,Y 509.902,Z 307.966,A -85,B 0,C 180,E1 -5572.078,E2 -5572.078} C_VEL
LIN {X 0,Y 509.956,Z 307.955,A -85,B 0,C 180,E1 -5574.464,E2 -5574.464} C_VEL
LIN {X 0,Y 510.031,Z 307.957,A -85,B 0,C 180,E1 -5577.631,E2 -5577.631} C_VEL
LIN {X 0,Y 510.022,Z 307.948,A -85,B 0,C 180,E1 -5580,E2 -5580} C_VEL
LIN {X 0,Y 510.034,Z 307.947,A -85,B 0,C 180,E1 -5582.369,E2 -5582.369} C_VEL
LIN {X 0,Y 509.931,Z 307.968,A -85,B 0,C 180,E1 -5585.536,E2 -5585.536} C_VEL
LIN {X 0,Y 509.891,Z 307.962,A -85,B 0,C 180,E1 -5588.721,E2 -5588.721} C_VEL
LIN {X 0,Y 509.896,Z 307.968,A -85,B 0,C 180,E1 -5591.932,E2 -5591.932} C_VEL
LIN {X 0,Y 509.887,Z 307.964,A -85,B 0,C 180,E1 -5595.242,E2 -5595.242} C_VEL
LIN {X 0,Y 509.829,Z 307.973,A -85,B 0,C 180,E1 -5598.485,E2 -5598.485} C_VEL
LIN {X 0,Y 509.836,Z 307.97,A -85,B 0,C 180,E1 -5601.002,E2 -5601.002} C_VEL
LIN {X 0,Y 509.81,Z 307.985,A -85,B 0,C 180,E1 -5603.565,E2 -5603.565} C_VEL
LIN {X 0,Y 509.81,Z 307.973,A -85,B 0,C 180,E1 -5606.357,E2 -5606.357} C_VEL
LIN {X 0,Y 509.829,Z 307.962,A -85,B 0,C 180,E1 -5608.847,E2 -5608.847} C_VEL
LIN {X 0,Y 509.811,Z 307.975,A -85,B 0,C 180,E1 -5611.591,E2 -5611.591} C_VEL
LIN {X 0,Y 509.828,Z 307.974,A -85,B 0,C 180,E1 -5614.415,E2 -5614.415} C_VEL
LIN {X 0,Y 509.8,Z 307.98,A -85,B 0,C 180,E1 -5617.342,E2 -5617.342} C_VEL
LIN {X 0,Y 509.807,Z 307.97,A -85,B 0,C 180,E1 -5620.386,E2 -5620.386} C_VEL
LIN {X 0,Y 509.801,Z 307.984,A -85,B 0,C 180,E1 -5623.574,E2 -5623.574} C_VEL
LIN {X 0,Y 509.788,Z 307.971,A -85,B 0,C 180,E1 -5626.426,E2 -5626.426} C_VEL
LIN {X 0,Y 509.809,Z 307.982,A -85,B 0,C 180,E1 -5629.616,E2 -5629.616} C_VEL
LIN {X 0,Y 509.79,Z 307.974,A -85,B 0,C 180,E1 -5632.658,E2 -5632.658} C_VEL
LIN {X 0,Y 509.799,Z 307.982,A -85,B 0,C 180,E1 -5633.694,E2 -5633.694} C_VEL
LIN {X 0,Y 509.135,Z 308.061,A -85,B 0,C 180,E1 -5634.353,E2 -5634.353} C_VEL
LIN {X 0,Y 506.319,Z 308.418,A -85,B 0,C 180,E1 -5635.425,E2 -5635.425} C_VEL
LIN {X 0,Y 503.926,Z 308.716,A -85,B 0,C 180,E1 -5636.289,E2 -5636.289} C_VEL
LIN {X 0,Y 502.876,Z 308.843,A -85,B 0,C 180,E1 -5636.955,E2 -5636.955} C_VEL
LIN {X 0,Y 502.779,Z 308.854,A -85,B 0,C 180,E1 -5637.181,E2 -5637.181} C_VEL
LIN {X 0,Y 502.789,Z 308.851,A -85,B 0,C 180,E1 -5640.071,E2 -5640.071} C_VEL
LIN {X 0,Y 502.77,Z 308.841,A -85,B 0,C 180,E1 -5642.53,E2 -5642.53} C_VEL
LIN {X 0,Y 502.762,Z 308.864,A -85,B 0,C 180,E1 -5645.316,E2 -5645.316} C_VEL
LIN {X 0,Y 502.779,Z 308.848,A -85,B 0,C 180,E1 -5647.827,E2 -5647.827} C_VEL
LIN {X 0,Y 502.806,Z 308.85,A -85,B 0,C 180,E1 -5650.4,E2 -5650.4} C_VEL
LIN {X 0,Y 502.774,Z 308.821,A -85,B 0,C 180,E1 -5652.93,E2 -5652.93} C_VEL
LIN {X 0,Y 502.846,Z 309.009,A -85,B 0,C 180,E1 -5654.497,E2 -5654.497} C_VEL
LIN {X 0,Y 503.114,Z 310.13,A -85,B 0,C 180,E1 -5654.638,E2 -5654.638} C_VEL
LIN {X 0,Y 505.452,Z 316.666,A -85,B 0,C 180,E1 -5654.821,E2 -5654.821} C_VEL
LIN {X 0,Y 505.19,Z 389.356,A -85,B 0,C 180,E1 -5655.884,E2 -5655.884} C_VEL
LIN {X 0,Y 505.095,Z 402.449,A -85,B 0,C 180,E1 -5656.241,E2 -5656.241} C_VEL
LIN {X 0,Y 504.918,Z 415.346,A -85,B 0,C 180,E1 -5656.764,E2 -5656.764} C_VEL
LIN {X 0,Y 504.72,Z 426.935,A -85,B 0,C 180,E1 -5657.408,E2 -5657.408} C_VEL
LIN {X 0,Y 504.304,Z 438.6,A -85,B 0,C 180,E1 -5658.24,E2 -5658.24} C_VEL
LIN {X 0,Y 503.984,Z 448.725,A -85,B 0,C 180,E1 -5659.149,E2 -5659.149} C_VEL
LIN {X 0,Y 503.691,Z 457.793,A -85,B 0,C 180,E1 -5660.159,E2 -5660.159} C_VEL
LIN {X 0,Y 503.333,Z 466.579,A -85,B 0,C 180,E1 -5661.367,E2 -5661.367} C_VEL
LIN {X 0,Y 503.123,Z 472.765,A -85,B 0,C 180,E1 -5662.415,E2 -5662.415} C_VEL
LIN {X 0,Y 502.971,Z 478.386,A -85,B 0,C 180,E1 -5663.582,E2 -5663.582} C_VEL
LIN {X 0,Y 502.704,Z 483.018,A -85,B 0,C 180,E1 -5664.786,E2 -5664.786} C_VEL
LIN {X 0,Y 502.618,Z 486.546,A -85,B 0,C 180,E1 -5665.991,E2 -5665.991} C_VEL
LIN {X 0,Y 502.544,Z 488.373,A -85,B 0,C 180,E1 -5666.793,E2 -5666.793} C_VEL
LIN {X 0,Y 502.556,Z 489.742,A -85,B 0,C 180,E1 -5667.596,E2 -5667.596} C_VEL
LIN {X 0,Y 502.52,Z 491.32,A -85,B 0,C 180,E1 -5669.199,E2 -5669.199} C_VEL
LIN {X 0,Y 502.506,Z 491.553,A -85,B 0,C 180,E1 -5670,E2 -5670} C_VEL
LIN {X 0,Y 502.519,Z 491.372,A -85,B 0,C 180,E1 -5670.801,E2 -5670.801} C_VEL
LIN {X 0,Y 502.556,Z 489.861,A -85,B 0,C 180,E1 -5672.404,E2 -5672.404} C_VEL
LIN {X 0,Y 502.54,Z 488.546,A -85,B 0,C 180,E1 -5673.207,E2 -5673.207} C_VEL
LIN {X 0,Y 502.683,Z 485.738,A -85,B 0,C 180,E1 -5674.41,E2 -5674.41} C_VEL
LIN {X 0,Y 502.856,Z 481.93,A -85,B 0,C 180,E1 -5675.614,E2 -5675.614} C_VEL
LIN {X 0,Y 502.936,Z 476.835,A -85,B 0,C 180,E1 -5676.866,E2 -5676.866} C_VEL
LIN {X 0,Y 503.239,Z 469.634,A -85,B 0,C 180,E1 -5678.23,E2 -5678.23} C_VEL
LIN {X 0,Y 503.556,Z 461.617,A -85,B 0,C 180,E1 -5679.438,E2 -5679.438} C_VEL
LIN {X 0,Y 503.839,Z 453.399,A -85,B 0,C 180,E1 -5680.447,E2 -5680.447} C_VEL
LIN {X 0,Y 504.151,Z 444.379,A -85,B 0,C 180,E1 -5681.356,E2 -5681.356} C_VEL
LIN {X 0,Y 504.542,Z 433.895,A -85,B 0,C 180,E1 -5682.208,E2 -5682.208} C_VEL
LIN {X 0,Y 504.75,Z 422.411,A -85,B 0,C 180,E1 -5682.955,E2 -5682.955} C_VEL
LIN {X 0,Y 504.982,Z 409.883,A -85,B 0,C 180,E1 -5683.573,E2 -5683.573} C_VEL
LIN {X 0,Y 505.141,Z 397.138,A -85,B 0,C 180,E1 -5684.015,E2 -5684.015} C_VEL
LIN {X 0,Y 505.169,Z 384.391,A -85,B 0,C 180,E1 -5684.296,E2 -5684.296} C_VEL
LIN {X 0,Y 505.414,Z 316.602,A -85,B 0,C 180,E1 -5685.272,E2 -5685.272} C_VEL
LIN {X 0,Y 502.928,Z 309.665,A -85,B 0,C 180,E1 -5685.486,E2 -5685.486} C_VEL
LIN {X 0,Y 502.81,Z 308.927,A -85,B 0,C 180,E1 -5685.635,E2 -5685.635} C_VEL
LIN {X 0,Y 502.799,Z 308.829,A -85,B 0,C 180,E1 -5688.753,E2 -5688.753} C_VEL
LIN {X 0,Y 502.773,Z 308.852,A -85,B 0,C 180,E1 -5691.311,E2 -5691.311} C_VEL
LIN {X 0,Y 502.755,Z 308.855,A -85,B 0,C 180,E1 -5693.915,E2 -5693.915} C_VEL
LIN {X 0,Y 502.756,Z 308.85,A -85,B 0,C 180,E1 -5696.572,E2 -5696.572} C_VEL
LIN {X 0,Y 502.788,Z 308.852,A -85,B 0,C 180,E1 -5699.29,E2 -5699.29} C_VEL
LIN {X 0,Y 502.754,Z 308.855,A -85,B 0,C 180,E1 -5702.086,E2 -5702.086} C_VEL
LIN {X 0,Y 502.784,Z 308.857,A -85,B 0,C 180,E1 -5704.966,E2 -5704.966} C_VEL
LIN {X 0,Y 502.76,Z 308.849,A -85,B 0,C 180,E1 -5707.956,E2 -5707.956} C_VEL
LIN {X 0,Y 502.758,Z 308.856,A -85,B 0,C 180,E1 -5711.071,E2 -5711.071} C_VEL
LIN {X 0,Y 502.774,Z 308.852,A -85,B 0,C 180,E1 -5714.528,E2 -5714.528} C_VEL
LIN {X 0,Y 502.761,Z 308.855,A -85,B 0,C 180,E1 -5717.857,E2 -5717.857} C_VEL
LIN {X 0,Y 502.777,Z 308.845,A -85,B 0,C 180,E1 -5721.021,E2 -5721.021} C_VEL
LIN {X 0,Y 502.76,Z 308.855,A -85,B 0,C 180,E1 -5724.17,E2 -5724.17} C_VEL
LIN {X 0,Y 502.797,Z 308.849,A -85,B 0,C 180,E1 -5726.998,E2 -5726.998} C_VEL
LIN {X 0,Y 502.784,Z 308.84,A -85,B 0,C 180,E1 -5730.069,E2 -5730.069} C_VEL
LIN {X 0,Y 502.777,Z 308.848,A -85,B 0,C 180,E1 -5733.429,E2 -5733.429} C_VEL
LIN {X 0,Y 502.752,Z 308.858,A -85,B 0,C 180,E1 -5736.084,E2 -5736.084} C_VEL
LIN {X 0,Y 502.761,Z 308.855,A -85,B 0,C 180,E1 -5738.688,E2 -5738.688} C_VEL
LIN {X 0,Y 502.798,Z 308.85,A -85,B 0,C 180,E1 -5741.247,E2 -5741.247} C_VEL
LIN {X 0,Y 502.827,Z 308.845,A -85,B 0,C 180,E1 -5744.664,E2 -5744.664} C_VEL
LIN {X 0,Y 502.868,Z 308.843,A -85,B 0,C 180,E1 -5748.039,E2 -5748.039} C_VEL
LIN {X 0,Y 502.831,Z 308.842,A -85,B 0,C 180,E1 -5751.156,E2 -5751.156} C_VEL
LIN {X 0,Y 502.839,Z 308.842,A -85,B 0,C 180,E1 -5753.58,E2 -5753.58} C_VEL
LIN {X 0,Y 502.855,Z 308.844,A -85,B 0,C 180,E1 -5756.795,E2 -5756.795} C_VEL
LIN {X 0,Y 502.89,Z 308.839,A -85,B 0,C 180,E1 -5758.398,E2 -5758.398} C_VEL
LIN {X 0,Y 502.98,Z 308.828,A -85,B 0,C 180,E1 -5760.801,E2 -5760.801} C_VEL
LIN {X 0,Y 502.998,Z 308.832,A -85,B 0,C 180,E1 -5762.402,E2 -5762.402} C_VEL
LIN {X 0,Y 502.909,Z 308.832,A -85,B 0,C 180,E1 -5765.614,E2 -5765.614} C_VEL
LIN {X 0,Y 502.863,Z 308.843,A -85,B 0,C 180,E1 -5768.034,E2 -5768.034} C_VEL
LIN {X 0,Y 502.828,Z 308.844,A -85,B 0,C 180,E1 -5771.284,E2 -5771.284} C_VEL
LIN {X 0,Y 502.833,Z 308.849,A -85,B 0,C 180,E1 -5774.571,E2 -5774.571} C_VEL
LIN {X 0,Y 502.792,Z 308.854,A -85,B 0,C 180,E1 -5777.91,E2 -5777.91} C_VEL
LIN {X 0,Y 502.822,Z 308.841,A -85,B 0,C 180,E1 -5780.536,E2 -5780.536} C_VEL
LIN {X 0,Y 502.779,Z 308.85,A -85,B 0,C 180,E1 -5783.041,E2 -5783.041} C_VEL
LIN {X 0,Y 502.77,Z 308.856,A -85,B 0,C 180,E1 -5785.679,E2 -5785.679} C_VEL
LIN {X 0,Y 502.787,Z 308.85,A -85,B 0,C 180,E1 -5788.376,E2 -5788.376} C_VEL
LIN {X 0,Y 502.788,Z 308.851,A -85,B 0,C 180,E1 -5791.144,E2 -5791.144} C_VEL
LIN {X 0,Y 502.78,Z 308.855,A -85,B 0,C 180,E1 -5793.996,E2 -5793.996} C_VEL
LIN {X 0,Y 502.727,Z 308.859,A -85,B 0,C 180,E1 -5797.171,E2 -5797.171} C_VEL
LIN {X 0,Y 502.765,Z 308.857,A -85,B 0,C 180,E1 -5800.018,E2 -5800.018} C_VEL
LIN {X 0,Y 502.745,Z 308.854,A -85,B 0,C 180,E1 -5803.234,E2 -5803.234} C_VEL
LIN {X 0,Y 502.762,Z 308.845,A -85,B 0,C 180,E1 -5805.659,E2 -5805.659} C_VEL
LIN {X 0,Y 502.76,Z 308.853,A -85,B 0,C 180,E1 -5809.013,E2 -5809.013} C_VEL
LIN {X 0,Y 502.757,Z 308.862,A -85,B 0,C 180,E1 -5812.044,E2 -5812.044} C_VEL
LIN {X 0,Y 502.78,Z 308.852,A -85,B 0,C 180,E1 -5815.033,E2 -5815.033} C_VEL
LIN {X 0,Y 502.776,Z 308.857,A -85,B 0,C 180,E1 -5817.915,E2 -5817.915} C_VEL
LIN {X 0,Y 502.856,Z 308.986,A -85,B 0,C 180,E1 -5820.959,E2 -5820.959} C_VEL
LIN {X 0,Y 505.619,Z 322.247,A -85,B 0,C 180,E1 -5822.822,E2 -5822.822} C_VEL
LIN {X 0,Y 505.058,Z 345.828,A -85,B 0,C 180,E1 -5825.764,E2 -5825.764} C_VEL
LIN {X 0,Y 504.357,Z 372.332,A -85,B 0,C 180,E1 -5829.006,E2 -5829.006} C_VEL
LIN {X 0,Y 503.721,Z 399.733,A -85,B 0,C 180,E1 -5832.335,E2 -5832.335} C_VEL
LIN {X 0,Y 503.393,Z 414.87,A -85,B 0,C 180,E1 -5834.152,E2 -5834.152} C_VEL
LIN {X 0,Y 505.245,Z 432.585,A -85,B 0,C 180,E1 -5834.485,E2 -5834.485} C_VEL
LIN {X 0,Y 504.75,Z 525.338,A -85,B 0,C 180,E1 -5835.82,E2 -5835.82} C_VEL
LIN {X 0,Y 504.442,Z 538.689,A -85,B 0,C 180,E1 -5836.171,E2 -5836.171} C_VEL
LIN {X 0,Y 504.075,Z 552.085,A -85,B 0,C 180,E1 -5836.7,E2 -5836.7} C_VEL
LIN {X 0,Y 503.689,Z 564.556,A -85,B 0,C 180,E1 -5837.382,E2 -5837.382} C_VEL
LIN {X 0,Y 503.387,Z 576.432,A -85,B 0,C 180,E1 -5838.218,E2 -5838.218} C_VEL
LIN {X 0,Y 503.035,Z 586.788,A -85,B 0,C 180,E1 -5839.128,E2 -5839.128} C_VEL
LIN {X 0,Y 502.747,Z 596.128,A -85,B 0,C 180,E1 -5840.14,E2 -5840.14} C_VEL
LIN {X 0,Y 502.507,Z 605.249,A -85,B 0,C 180,E1 -5841.353,E2 -5841.353} C_VEL
LIN {X 0,Y 502.364,Z 612.611,A -85,B 0,C 180,E1 -5842.565,E2 -5842.565} C_VEL
LIN {X 0,Y 502.303,Z 617.591,A -85,B 0,C 180,E1 -5843.573,E2 -5843.573} C_VEL
LIN {X 0,Y 502.279,Z 622.44,A -85,B 0,C 180,E1 -5844.782,E2 -5844.782} C_VEL
LIN {X 0,Y 502.342,Z 626.158,A -85,B 0,C 180,E1 -5845.989,E2 -5845.989} C_VEL
LIN {X 0,Y 502.26,Z 628.062,A -85,B 0,C 180,E1 -5846.791,E2 -5846.791} C_VEL
LIN {X 0,Y 502.221,Z 629.493,A -85,B 0,C 180,E1 -5847.594,E2 -5847.594} C_VEL
LIN {X 0,Y 502.233,Z 631.145,A -85,B 0,C 180,E1 -5849.198,E2 -5849.198} C_VEL
LIN {X 0,Y 502.225,Z 631.366,A -85,B 0,C 180,E1 -5850,E2 -5850} C_VEL
LIN {X 0,Y 502.233,Z 631.145,A -85,B 0,C 180,E1 -5850.802,E2 -5850.802} C_VEL
LIN {X 0,Y 502.221,Z 629.496,A -85,B 0,C 180,E1 -5852.406,E2 -5852.406} C_VEL
LIN {X 0,Y 502.26,Z 628.066,A -85,B 0,C 180,E1 -5853.209,E2 -5853.209} C_VEL
LIN {X 0,Y 502.273,Z 625.05,A -85,B 0,C 180,E1 -5854.414,E2 -5854.414} C_VEL
LIN {X 0,Y 502.286,Z 620.969,A -85,B 0,C 180,E1 -5855.621,E2 -5855.621} C_VEL
LIN {X 0,Y 502.337,Z 614.804,A -85,B 0,C 180,E1 -5857.011,E2 -5857.011} C_VEL
LIN {X 0,Y 502.471,Z 607.871,A -85,B 0,C 180,E1 -5858.242,E2 -5858.242} C_VEL
LIN {X 0,Y 502.627,Z 599.409,A -85,B 0,C 180,E1 -5859.456,E2 -5859.456} C_VEL
LIN {X 0,Y 502.874,Z 590.758,A -85,B 0,C 180,E1 -5860.468,E2 -5860.468} C_VEL
LIN {X 0,Y 503.202,Z 580.099,A -85,B 0,C 180,E1 -5861.48,E2 -5861.48} C_VEL
LIN {X 0,Y 503.525,Z 569.389,A -85,B 0,C 180,E1 -5862.303,E2 -5862.303} C_VEL
LIN {X 0,Y 503.86,Z 558.072,A -85,B 0,C 180,E1 -5862.998,E2 -5862.998} C_VEL
LIN {X 0,Y 504.262,Z 546.303,A -85,B 0,C 180,E1 -5863.551,E2 -5863.551} C_VEL
LIN {X 0,Y 504.595,Z 532.778,A -85,B 0,C 180,E1 -5864.004,E2 -5864.004} C_VEL
LIN {X 0,Y 504.829,Z 519.451,A -85,B 0,C 180,E1 -5864.28,E2 -5864.28} C_VEL
LIN {X 0,Y 505.156,Z 431.102,A -85,B 0,C 180,E1 -5865.539,E2 -5865.539} C_VEL
LIN {X 0,Y 503.39,Z 414.921,A -85,B 0,C 180,E1 -5865.845,E2 -5865.845} C_VEL
LIN {X 0,Y 503.944,Z 389.395,A -85,B 0,C 180,E1 -5868.919,E2 -5868.919} C_VEL
LIN {X 0,Y 504.57,Z 363.324,A -85,B 0,C 180,E1 -5872.09,E2 -5872.09} C_VEL
LIN {X 0,Y 505.287,Z 337.215,A -85,B 0,C 180,E1 -5875.3,E2 -5875.3} C_VEL
LIN {X 0,Y 505.619,Z 322.231,A -85,B 0,C 180,E1 -5877.178,E2 -5877.178} C_VEL
LIN {X 0,Y 502.834,Z 308.96,A -85,B 0,C 180,E1 -5879.057,E2 -5879.057} C_VEL
LIN {X 0,Y 502.776,Z 308.857,A -85,B 0,C 180,E1 -5882.084,E2 -5882.084} C_VEL
LIN {X 0,Y 502.781,Z 308.853,A -85,B 0,C 180,E1 -5884.967,E2 -5884.967} C_VEL
LIN {X 0,Y 502.76,Z 308.854,A -85,B 0,C 180,E1 -5888.481,E2 -5888.481} C_VEL
LIN {X 0,Y 502.759,Z 308.854,A -85,B 0,C 180,E1 -5891.071,E2 -5891.071} C_VEL
LIN {X 0,Y 502.781,Z 308.841,A -85,B 0,C 180,E1 -5894.529,E2 -5894.529} C_VEL
LIN {X 0,Y 502.761,Z 308.86,A -85,B 0,C 180,E1 -5897.857,E2 -5897.857} C_VEL
LIN {X 0,Y 502.777,Z 308.846,A -85,B 0,C 180,E1 -5901.022,E2 -5901.022} C_VEL
LIN {X 0,Y 502.751,Z 308.847,A -85,B 0,C 180,E1 -5904.171,E2 -5904.171} C_VEL
LIN {X 0,Y 502.797,Z 308.849,A -85,B 0,C 180,E1 -5906.998,E2 -5906.998} C_VEL
LIN {X 0,Y 502.809,Z 308.849,A -85,B 0,C 180,E1 -5910.064,E2 -5910.064} C_VEL
LIN {X 0,Y 502.779,Z 308.85,A -85,B 0,C 180,E1 -5912.53,E2 -5912.53} C_VEL
LIN {X 0,Y 502.763,Z 308.856,A -85,B 0,C 180,E1 -5915.313,E2 -5915.313} C_VEL
LIN {X 0,Y 502.772,Z 308.853,A -85,B 0,C 180,E1 -5917.826,E2 -5917.826} C_VEL
LIN {X 0,Y 502.811,Z 308.844,A -85,B 0,C 180,E1 -5920.4,E2 -5920.4} C_VEL
LIN {X 0,Y 502.801,Z 308.849,A -85,B 0,C 180,E1 -5922.93,E2 -5922.93} C_VEL
LIN {X 0,Y 502.833,Z 308.849,A -85,B 0,C 180,E1 -5925.429,E2 -5925.429} C_VEL
LIN {X 0,Y 502.866,Z 308.84,A -85,B 0,C 180,E1 -5928.717,E2 -5928.717} C_VEL
LIN {X 0,Y 502.863,Z 308.844,A -85,B 0,C 180,E1 -5931.966,E2 -5931.966} C_VEL
LIN {X 0,Y 502.91,Z 308.833,A -85,B 0,C 180,E1 -5934.386,E2 -5934.386} C_VEL
LIN {X 0,Y 502.999,Z 308.832,A -85,B 0,C 180,E1 -5937.598,E2 -5937.598} C_VEL
LIN {X 0,Y 502.991,Z 308.823,A -85,B 0,C 180,E1 -5940,E2 -5940} C_VEL
LIN {X 0,Y 503.004,Z 308.823,A -85,B 0,C 180,E1 -5942.402,E2 -5942.402} C_VEL
LIN {X 0,Y 502.888,Z 308.845,A -85,B 0,C 180,E1 -5945.614,E2 -5945.614} C_VEL
LIN {X 0,Y 502.862,Z 308.84,A -85,B 0,C 180,E1 -5948.034,E2 -5948.034} C_VEL
LIN {X 0,Y 502.866,Z 308.844,A -85,B 0,C 180,E1 -5951.283,E2 -5951.283} C_VEL
LIN {X 0,Y 502.818,Z 308.84,A -85,B 0,C 180,E1 -5954.572,E2 -5954.572} C_VEL
LIN {X 0,Y 502.792,Z 308.854,A -85,B 0,C 180,E1 -5957.91,E2 -5957.91} C_VEL
LIN {X 0,Y 502.822,Z 308.842,A -85,B 0,C 180,E1 -5960.537,E2 -5960.537} C_VEL
LIN {X 0,Y 502.778,Z 308.853,A -85,B 0,C 180,E1 -5963.041,E2 -5963.041} C_VEL
LIN {X 0,Y 502.77,Z 308.856,A -85,B 0,C 180,E1 -5965.68,E2 -5965.68} C_VEL
LIN {X 0,Y 502.765,Z 308.841,A -85,B 0,C 180,E1 -5968.377,E2 -5968.377} C_VEL
LIN {X 0,Y 502.784,Z 308.847,A -85,B 0,C 180,E1 -5971.499,E2 -5971.499} C_VEL
LIN {X 0,Y 502.78,Z 308.852,A -85,B 0,C 180,E1 -5974.442,E2 -5974.442} C_VEL
LIN {X 0,Y 502.758,Z 308.857,A -85,B 0,C 180,E1 -5977.176,E2 -5977.176} C_VEL
LIN {X 0,Y 502.764,Z 308.849,A -85,B 0,C 180,E1 -5980.018,E2 -5980.018} C_VEL
LIN {X 0,Y 502.742,Z 308.863,A -85,B 0,C 180,E1 -5983.235,E2 -5983.235} C_VEL
LIN {X 0,Y 502.763,Z 308.851,A -85,B 0,C 180,E1 -5985.659,E2 -5985.659} C_VEL
LIN {X 0,Y 502.76,Z 308.856,A -85,B 0,C 180,E1 -5989.013,E2 -5989.013} C_VEL
LIN {X 0,Y 502.761,Z 308.85,A -85,B 0,C 180,E1 -5992.044,E2 -5992.044} C_VEL
LIN {X 0,Y 502.788,Z 308.855,A -85,B 0,C 180,E1 -5995.034,E2 -5995.034} C_VEL
LIN {X 0,Y 502.779,Z 308.854,A -85,B 0,C 180,E1 -5997.181,E2 -5997.181} C_VEL
LIN {X 0,Y 502.08,Z 308.941,A -85,B 0,C 180,E1 -5997.85,E2 -5997.85} C_VEL
LIN {X 0,Y 499.222,Z 309.298,A -85,B 0,C 180,E1 -5998.935,E2 -5998.935} C_VEL
LIN {X 0,Y 496.825,Z 309.596,A -85,B 0,C 180,E1 -5999.81,E2 -5999.81} C_VEL
LIN {X 0,Y 495.797,Z 309.722,A -85,B 0,C 180,E1 -6000.486,E2 -6000.486} C_VEL
LIN {X 0,Y 495.712,Z 309.73,A -85,B 0,C 180,E1 -6000.715,E2 -6000.715} C_VEL
LIN {X 0,Y 495.706,Z 309.734,A -85,B 0,C 180,E1 -6003.928,E2 -6003.928} C_VEL
LIN {X 0,Y 495.758,Z 309.725,A -85,B 0,C 180,E1 -6007.141,E2 -6007.141} C_VEL
LIN {X 0,Y 495.757,Z 309.729,A -85,B 0,C 180,E1 -6010.109,E2 -6010.109} C_VEL
LIN {X 0,Y 495.721,Z 309.698,A -85,B 0,C 180,E1 -6012.679,E2 -6012.679} C_VEL
LIN {X 0,Y 495.782,Z 309.895,A -85,B 0,C 180,E1 -6014.27,E2 -6014.27} C_VEL
LIN {X 0,Y 495.985,Z 310.814,A -85,B 0,C 180,E1 -6014.401,E2 -6014.401} C_VEL
LIN {X 0,Y 498.739,Z 318.88,A -85,B 0,C 180,E1 -6014.629,E2 -6014.629} C_VEL
LIN {X 0,Y 498.356,Z 390.358,A -85,B 0,C 180,E1 -6015.687,E2 -6015.687} C_VEL
LIN {X 0,Y 498.261,Z 403.442,A -85,B 0,C 180,E1 -6016.048,E2 -6016.048} C_VEL
LIN {X 0,Y 498.092,Z 415.453,A -85,B 0,C 180,E1 -6016.538,E2 -6016.538} C_VEL
LIN {X 0,Y 497.88,Z 426.735,A -85,B 0,C 180,E1 -6017.154,E2 -6017.154} C_VEL
LIN {X 0,Y 497.472,Z 438.313,A -85,B 0,C 180,E1 -6017.973,E2 -6017.973} C_VEL
LIN {X 0,Y 497.113,Z 448.661,A -85,B 0,C 180,E1 -6018.894,E2 -6018.894} C_VEL
LIN {X 0,Y 496.821,Z 457.098,A -85,B 0,C 180,E1 -6019.815,E2 -6019.815} C_VEL
LIN {X 0,Y 496.467,Z 464.866,A -85,B 0,C 180,E1 -6020.837,E2 -6020.837} C_VEL
LIN {X 0,Y 496.199,Z 472.549,A -85,B 0,C 180,E1 -6022.083,E2 -6022.083} C_VEL
LIN {X 0,Y 495.996,Z 478.31,A -85,B 0,C 180,E1 -6023.245,E2 -6023.245} C_VEL
LIN {X 0,Y 495.875,Z 482.592,A -85,B 0,C 180,E1 -6024.306,E2 -6024.306} C_VEL
LIN {X 0,Y 495.675,Z 486.481,A -85,B 0,C 180,E1 -6025.527,E2 -6025.527} C_VEL
LIN {X 0,Y 495.523,Z 489.353,A -85,B 0,C 180,E1 -6026.748,E2 -6026.748} C_VEL
LIN {X 0,Y 495.543,Z 490.72,A -85,B 0,C 180,E1 -6027.562,E2 -6027.562} C_VEL
LIN {X 0,Y 495.504,Z 492.296,A -85,B 0,C 180,E1 -6029.187,E2 -6029.187} C_VEL
LIN {X 0,Y 495.49,Z 492.529,A -85,B 0,C 180,E1 -6030,E2 -6030} C_VEL
LIN {X 0,Y 495.504,Z 492.348,A -85,B 0,C 180,E1 -6030.813,E2 -6030.813} C_VEL
LIN {X 0,Y 495.542,Z 490.837,A -85,B 0,C 180,E1 -6032.438,E2 -6032.438} C_VEL
LIN {X 0,Y 495.519,Z 489.523,A -85,B 0,C 180,E1 -6033.252,E2 -6033.252} C_VEL
LIN {X 0,Y 495.672,Z 486.715,A -85,B 0,C 180,E1 -6034.473,E2 -6034.473} C_VEL
LIN {X 0,Y 495.871,Z 482.905,A -85,B 0,C 180,E1 -6035.694,E2 -6035.694} C_VEL
LIN {X 0,Y 495.958,Z 477.816,A -85,B 0,C 180,E1 -6036.962,E2 -6036.962} C_VEL
LIN {X 0,Y 496.286,Z 470.609,A -85,B 0,C 180,E1 -6038.346,E2 -6038.346} C_VEL
LIN {X 0,Y 496.629,Z 462.591,A -85,B 0,C 180,E1 -6039.571,E2 -6039.571} C_VEL
LIN {X 0,Y 496.951,Z 454.37,A -85,B 0,C 180,E1 -6040.594,E2 -6040.594} C_VEL
LIN {X 0,Y 497.26,Z 445.352,A -85,B 0,C 180,E1 -6041.515,E2 -6041.515} C_VEL
LIN {X 0,Y 497.676,Z 434.867,A -85,B 0,C 180,E1 -6042.379,E2 -6042.379} C_VEL
LIN {X 0,Y 497.902,Z 423.381,A -85,B 0,C 180,E1 -6043.136,E2 -6043.136} C_VEL
LIN {X 0,Y 498.147,Z 410.85,A -85,B 0,C 180,E1 -6043.762,E2 -6043.762} C_VEL
LIN {X 0,Y 498.312,Z 398.101,A -85,B 0,C 180,E1 -6044.211,E2 -6044.211} C_VEL
LIN {X 0,Y 498.336,Z 385.344,A -85,B 0,C 180,E1 -6044.497,E2 -6044.497} C_VEL
LIN {X 0,Y 498.593,Z 318.181,A -85,B 0,C 180,E1 -6045.477,E2 -6045.477} C_VEL
LIN {X 0,Y 495.91,Z 310.572,A -85,B 0,C 180,E1 -6045.709,E2 -6045.709} C_VEL
LIN {X 0,Y 495.752,Z 309.807,A -85,B 0,C 180,E1 -6045.863,E2 -6045.863} C_VEL
LIN {X 0,Y 495.753,Z 309.713,A -85,B 0,C 180,E1 -6049.029,E2 -6049.029} C_VEL
LIN {X 0,Y 495.736,Z 309.727,A -85,B 0,C 180,E1 -6051.629,E2 -6051.629} C_VEL
LIN {X 0,Y 495.702,Z 309.736,A -85,B 0,C 180,E1 -6054.277,E2 -6054.277} C_VEL
LIN {X 0,Y 495.717,Z 309.72,A -85,B 0,C 180,E1 -6056.979,E2 -6056.979} C_VEL
LIN {X 0,Y 495.736,Z 309.73,A -85,B 0,C 180,E1 -6060.141,E2 -6060.141} C_VEL
LIN {X 0,Y 495.726,Z 309.732,A -85,B 0,C 180,E1 -6063.232,E2 -6063.232} C_VEL
LIN {X 0,Y 495.702,Z 309.735,A -85,B 0,C 180,E1 -6066.085,E2 -6066.085} C_VEL
LIN {X 0,Y 495.736,Z 309.734,A -85,B 0,C 180,E1 -6068.764,E2 -6068.764} C_VEL
LIN {X 0,Y 495.72,Z 309.729,A -85,B 0,C 180,E1 -6071.784,E2 -6071.784} C_VEL
LIN {X 0,Y 495.727,Z 309.733,A -85,B 0,C 180,E1 -6075.141,E2 -6075.141} C_VEL
LIN {X 0,Y 495.718,Z 309.735,A -85,B 0,C 180,E1 -6078.215,E2 -6078.215} C_VEL
LIN {X 0,Y 495.735,Z 309.72,A -85,B 0,C 180,E1 -6081.235,E2 -6081.235} C_VEL
LIN {X 0,Y 495.733,Z 309.735,A -85,B 0,C 180,E1 -6084.461,E2 -6084.461} C_VEL
LIN {X 0,Y 495.744,Z 309.725,A -85,B 0,C 180,E1 -6087.404,E2 -6087.404} C_VEL
LIN {X 0,Y 495.733,Z 309.717,A -85,B 0,C 180,E1 -6090.251,E2 -6090.251} C_VEL
LIN {X 0,Y 495.732,Z 309.726,A -85,B 0,C 180,E1 -6093.27,E2 -6093.27} C_VEL
LIN {X 0,Y 495.701,Z 309.734,A -85,B 0,C 180,E1 -6095.722,E2 -6095.722} C_VEL
LIN {X 0,Y 495.724,Z 309.735,A -85,B 0,C 180,E1 -6098.37,E2 -6098.37} C_VEL
LIN {X 0,Y 495.756,Z 309.729,A -85,B 0,C 180,E1 -6100.97,E2 -6100.97} C_VEL
LIN {X 0,Y 495.814,Z 309.72,A -85,B 0,C 180,E1 -6104.549,E2 -6104.549} C_VEL
LIN {X 0,Y 495.82,Z 309.72,A -85,B 0,C 180,E1 -6107.965,E2 -6107.965} C_VEL
LIN {X 0,Y 495.789,Z 309.719,A -85,B 0,C 180,E1 -6111.029,E2 -6111.029} C_VEL
LIN {X 0,Y 495.795,Z 309.719,A -85,B 0,C 180,E1 -6113.488,E2 -6113.488} C_VEL
LIN {X 0,Y 495.711,Z 309.735,A -85,B 0,C 180,E1 -6115.935,E2 -6115.935} C_VEL
LIN {X 0,Y 495.972,Z 309.699,A -85,B 0,C 180,E1 -6117.564,E2 -6117.564} C_VEL
LIN {X 0,Y 495.932,Z 309.706,A -85,B 0,C 180,E1 -6120.812,E2 -6120.812} C_VEL
LIN {X 0,Y 495.965,Z 309.708,A -85,B 0,C 180,E1 -6122.436,E2 -6122.436} C_VEL
LIN {X 0,Y 495.866,Z 309.71,A -85,B 0,C 180,E1 -6125.694,E2 -6125.694} C_VEL
LIN {X 0,Y 495.819,Z 309.722,A -85,B 0,C 180,E1 -6128.149,E2 -6128.149} C_VEL
LIN {X 0,Y 495.812,Z 309.718,A -85,B 0,C 180,E1 -6131.446,E2 -6131.446} C_VEL
LIN {X 0,Y 495.779,Z 309.726,A -85,B 0,C 180,E1 -6134.783,E2 -6134.783} C_VEL
LIN {X 0,Y 495.771,Z 309.729,A -85,B 0,C 180,E1 -6138.172,E2 -6138.172} C_VEL
LIN {X 0,Y 495.767,Z 309.718,A -85,B 0,C 180,E1 -6140.757,E2 -6140.757} C_VEL
LIN {X 0,Y 495.731,Z 309.728,A -85,B 0,C 180,E1 -6143.388,E2 -6143.388} C_VEL
LIN {X 0,Y 495.732,Z 309.728,A -85,B 0,C 180,E1 -6146.73,E2 -6146.73} C_VEL
LIN {X 0,Y 495.756,Z 309.725,A -85,B 0,C 180,E1 -6149.747,E2 -6149.747} C_VEL
LIN {X 0,Y 495.746,Z 309.729,A -85,B 0,C 180,E1 -6152.596,E2 -6152.596} C_VEL
LIN {X 0,Y 495.722,Z 309.729,A -85,B 0,C 180,E1 -6155.54,E2 -6155.54} C_VEL
LIN {X 0,Y 495.734,Z 309.727,A -85,B 0,C 180,E1 -6158.765,E2 -6158.765} C_VEL
LIN {X 0,Y 495.72,Z 309.737,A -85,B 0,C 180,E1 -6161.785,E2 -6161.785} C_VEL
LIN {X 0,Y 495.728,Z 309.717,A -85,B 0,C 180,E1 -6165.142,E2 -6165.142} C_VEL
LIN {X 0,Y 495.719,Z 309.737,A -85,B 0,C 180,E1 -6168.216,E2 -6168.216} C_VEL
LIN {X 0,Y 495.736,Z 309.727,A -85,B 0,C 180,E1 -6171.236,E2 -6171.236} C_VEL
LIN {X 0,Y 495.726,Z 309.731,A -85,B 0,C 180,E1 -6174.461,E2 -6174.461} C_VEL
LIN {X 0,Y 495.748,Z 309.727,A -85,B 0,C 180,E1 -6177.405,E2 -6177.405} C_VEL
LIN {X 0,Y 495.826,Z 309.908,A -85,B 0,C 180,E1 -6180.754,E2 -6180.754} C_VEL
LIN {X 0,Y 498.616,Z 323.012,A -85,B 0,C 180,E1 -6182.622,E2 -6182.622} C_VEL
LIN {X 0,Y 498.575,Z 330.919,A -85,B 0,C 180,E1 -6183.639,E2 -6183.639} C_VEL
LIN {X 0,Y 497.843,Z 354.318,A -85,B 0,C 180,E1 -6186.578,E2 -6186.578} C_VEL
LIN {X 0,Y 497.2,Z 378.095,A -85,B 0,C 180,E1 -6189.523,E2 -6189.523} C_VEL
LIN {X 0,Y 496.561,Z 403.935,A -85,B 0,C 180,E1 -6192.71,E2 -6192.71} C_VEL
LIN {X 0,Y 496.348,Z 413.839,A -85,B 0,C 180,E1 -6193.918,E2 -6193.918} C_VEL
LIN {X 0,Y 498.387,Z 433.178,A -85,B 0,C 180,E1 -6194.289,E2 -6194.289} C_VEL
LIN {X 0,Y 497.867,Z 524.35,A -85,B 0,C 180,E1 -6195.62,E2 -6195.62} C_VEL
LIN {X 0,Y 497.513,Z 537.696,A -85,B 0,C 180,E1 -6195.975,E2 -6195.975} C_VEL
LIN {X 0,Y 497.191,Z 549.962,A -85,B 0,C 180,E1 -6196.461,E2 -6196.461} C_VEL
LIN {X 0,Y 496.744,Z 562.369,A -85,B 0,C 180,E1 -6197.125,E2 -6197.125} C_VEL
LIN {X 0,Y 496.42,Z 574.124,A -85,B 0,C 180,E1 -6197.947,E2 -6197.947} C_VEL
LIN {X 0,Y 495.933,Z 584.71,A -85,B 0,C 180,E1 -6198.867,E2 -6198.867} C_VEL
LIN {X 0,Y 495.727,Z 593.413,A -85,B 0,C 180,E1 -6199.793,E2 -6199.793} C_VEL
LIN {X 0,Y 495.496,Z 601.452,A -85,B 0,C 180,E1 -6200.818,E2 -6200.818} C_VEL
LIN {X 0,Y 495.343,Z 609.33,A -85,B 0,C 180,E1 -6202.049,E2 -6202.049} C_VEL
LIN {X 0,Y 495.252,Z 616.603,A -85,B 0,C 180,E1 -6203.481,E2 -6203.481} C_VEL
LIN {X 0,Y 495.21,Z 621.452,A -85,B 0,C 180,E1 -6204.707,E2 -6204.707} C_VEL
LIN {X 0,Y 495.296,Z 625.176,A -85,B 0,C 180,E1 -6205.932,E2 -6205.932} C_VEL
LIN {X 0,Y 495.215,Z 627.08,A -85,B 0,C 180,E1 -6206.746,E2 -6206.746} C_VEL
LIN {X 0,Y 495.179,Z 628.512,A -85,B 0,C 180,E1 -6207.56,E2 -6207.56} C_VEL
LIN {X 0,Y 495.216,Z 630.168,A -85,B 0,C 180,E1 -6209.187,E2 -6209.187} C_VEL
LIN {X 0,Y 495.206,Z 630.39,A -85,B 0,C 180,E1 -6210,E2 -6210} C_VEL
LIN {X 0,Y 495.216,Z 630.169,A -85,B 0,C 180,E1 -6210.813,E2 -6210.813} C_VEL
LIN {X 0,Y 495.179,Z 628.516,A -85,B 0,C 180,E1 -6212.44,E2 -6212.44} C_VEL
LIN {X 0,Y 495.214,Z 627.084,A -85,B 0,C 180,E1 -6213.254,E2 -6213.254} C_VEL
LIN {X 0,Y 495.216,Z 624.066,A -85,B 0,C 180,E1 -6214.477,E2 -6214.477} C_VEL
LIN {X 0,Y 495.23,Z 619.983,A -85,B 0,C 180,E1 -6215.701,E2 -6215.701} C_VEL
LIN {X 0,Y 495.272,Z 613.814,A -85,B 0,C 180,E1 -6217.112,E2 -6217.112} C_VEL
LIN {X 0,Y 495.416,Z 606.879,A -85,B 0,C 180,E1 -6218.361,E2 -6218.361} C_VEL
LIN {X 0,Y 495.569,Z 598.413,A -85,B 0,C 180,E1 -6219.592,E2 -6219.592} C_VEL
LIN {X 0,Y 495.835,Z 589.762,A -85,B 0,C 180,E1 -6220.618,E2 -6220.618} C_VEL
LIN {X 0,Y 496.211,Z 579.106,A -85,B 0,C 180,E1 -6221.644,E2 -6221.644} C_VEL
LIN {X 0,Y 496.588,Z 567.793,A -85,B 0,C 180,E1 -6222.521,E2 -6222.521} C_VEL
LIN {X 0,Y 496.874,Z 557.074,A -85,B 0,C 180,E1 -6223.184,E2 -6223.184} C_VEL
LIN {X 0,Y 497.311,Z 545.308,A -85,B 0,C 180,E1 -6223.744,E2 -6223.744} C_VEL
LIN {X 0,Y 497.688,Z 531.787,A -85,B 0,C 180,E1 -6224.203,E2 -6224.203} C_VEL
LIN {X 0,Y 497.94,Z 518.462,A -85,B 0,C 180,E1 -6224.482,E2 -6224.482} C_VEL
LIN {X 0,Y 498.284,Z 431.574,A -85,B 0,C 180,E1 -6225.738,E2 -6225.738} C_VEL
LIN {X 0,Y 496.362,Z 414.086,A -85,B 0,C 180,E1 -6226.066,E2 -6226.066} C_VEL
LIN {X 0,Y 496.928,Z 390.203,A -85,B 0,C 180,E1 -6228.983,E2 -6228.983} C_VEL
LIN {X 0,Y 497.598,Z 364.165,A -85,B 0,C 180,E1 -6232.198,E2 -6232.198} C_VEL
LIN {X 0,Y 498.329,Z 339.544,A -85,B 0,C 180,E1 -6235.269,E2 -6235.269} C_VEL
LIN {X 0,Y 498.78,Z 324.932,A -85,B 0,C 180,E1 -6237.121,E2 -6237.121} C_VEL
LIN {X 0,Y 497.707,Z 318.526,A -85,B 0,C 180,E1 -6238.001,E2 -6238.001} C_VEL
LIN {X 0,Y 495.812,Z 309.832,A -85,B 0,C 180,E1 -6239.276,E2 -6239.276} C_VEL
LIN {X 0,Y 495.748,Z 309.728,A -85,B 0,C 180,E1 -6242.595,E2 -6242.595} C_VEL
LIN {X 0,Y 495.727,Z 309.731,A -85,B 0,C 180,E1 -6245.539,E2 -6245.539} C_VEL
LIN {X 0,Y 495.737,Z 309.727,A -85,B 0,C 180,E1 -6248.764,E2 -6248.764} C_VEL
LIN {X 0,Y 495.719,Z 309.737,A -85,B 0,C 180,E1 -6251.784,E2 -6251.784} C_VEL
LIN {X 0,Y 495.733,Z 309.716,A -85,B 0,C 180,E1 -6255.14,E2 -6255.14} C_VEL
LIN {X 0,Y 495.72,Z 309.737,A -85,B 0,C 180,E1 -6258.215,E2 -6258.215} C_VEL
LIN {X 0,Y 495.734,Z 309.724,A -85,B 0,C 180,E1 -6261.235,E2 -6261.235} C_VEL
LIN {X 0,Y 495.727,Z 309.723,A -85,B 0,C 180,E1 -6264.46,E2 -6264.46} C_VEL
LIN {X 0,Y 495.746,Z 309.729,A -85,B 0,C 180,E1 -6267.404,E2 -6267.404} C_VEL
LIN {X 0,Y 495.757,Z 309.724,A -85,B 0,C 180,E1 -6270.253,E2 -6270.253} C_VEL
LIN {X 0,Y 495.733,Z 309.728,A -85,B 0,C 180,E1 -6273.27,E2 -6273.27} C_VEL
LIN {X 0,Y 495.731,Z 309.728,A -85,B 0,C 180,E1 -6276.612,E2 -6276.612} C_VEL
LIN {X 0,Y 495.771,Z 309.717,A -85,B 0,C 180,E1 -6279.324,E2 -6279.324} C_VEL
LIN {X 0,Y 495.771,Z 309.729,A -85,B 0,C 180,E1 -6281.828,E2 -6281.828} C_VEL
LIN {X 0,Y 495.779,Z 309.725,A -85,B 0,C 180,E1 -6285.217,E2 -6285.217} C_VEL
LIN {X 0,Y 495.841,Z 309.715,A -85,B 0,C 180,E1 -6288.555,E2 -6288.555} C_VEL
LIN {X 0,Y 495.82,Z 309.723,A -85,B 0,C 180,E1 -6291.851,E2 -6291.851} C_VEL
LIN {X 0,Y 495.867,Z 309.711,A -85,B 0,C 180,E1 -6294.306,E2 -6294.306} C_VEL
LIN {X 0,Y 495.966,Z 309.707,A -85,B 0,C 180,E1 -6297.564,E2 -6297.564} C_VEL
LIN {X 0,Y 495.961,Z 309.699,A -85,B 0,C 180,E1 -6300,E2 -6300} C_VEL
LIN {X 0,Y 495.972,Z 309.699,A -85,B 0,C 180,E1 -6302.436,E2 -6302.436} C_VEL
LIN {X 0,Y 495.846,Z 309.721,A -85,B 0,C 180,E1 -6305.694,E2 -6305.694} C_VEL
LIN {X 0,Y 495.821,Z 309.716,A -85,B 0,C 180,E1 -6308.149,E2 -6308.149} C_VEL
LIN {X 0,Y 495.842,Z 309.722,A -85,B 0,C 180,E1 -6311.446,E2 -6311.446} C_VEL
LIN {X 0,Y 495.768,Z 309.718,A -85,B 0,C 180,E1 -6314.784,E2 -6314.784} C_VEL
LIN {X 0,Y 495.771,Z 309.726,A -85,B 0,C 180,E1 -6318.172,E2 -6318.172} C_VEL
LIN {X 0,Y 495.767,Z 309.721,A -85,B 0,C 180,E1 -6320.757,E2 -6320.757} C_VEL
LIN {X 0,Y 495.731,Z 309.735,A -85,B 0,C 180,E1 -6323.388,E2 -6323.388} C_VEL
LIN {X 0,Y 495.732,Z 309.726,A -85,B 0,C 180,E1 -6326.73,E2 -6326.73} C_VEL
LIN {X 0,Y 495.735,Z 309.717,A -85,B 0,C 180,E1 -6329.749,E2 -6329.749} C_VEL
LIN {X 0,Y 495.745,Z 309.724,A -85,B 0,C 180,E1 -6332.596,E2 -6332.596} C_VEL
LIN {X 0,Y 495.737,Z 309.735,A -85,B 0,C 180,E1 -6335.539,E2 -6335.539} C_VEL
LIN {X 0,Y 495.737,Z 309.719,A -85,B 0,C 180,E1 -6338.766,E2 -6338.766} C_VEL
LIN {X 0,Y 495.718,Z 309.735,A -85,B 0,C 180,E1 -6341.785,E2 -6341.785} C_VEL
LIN {X 0,Y 495.729,Z 309.735,A -85,B 0,C 180,E1 -6345.142,E2 -6345.142} C_VEL
LIN {X 0,Y 495.72,Z 309.729,A -85,B 0,C 180,E1 -6348.216,E2 -6348.216} C_VEL
LIN {X 0,Y 495.736,Z 309.736,A -85,B 0,C 180,E1 -6351.236,E2 -6351.236} C_VEL
LIN {X 0,Y 495.739,Z 309.729,A -85,B 0,C 180,E1 -6354.462,E2 -6354.462} C_VEL
LIN {X 0,Y 495.739,Z 309.731,A -85,B 0,C 180,E1 -6357.404,E2 -6357.404} C_VEL
LIN {X 0,Y 495.738,Z 309.729,A -85,B 0,C 180,E1 -6360.252,E2 -6360.252} C_VEL
LIN {X 0,Y 495.712,Z 309.73,A -85,B 0,C 180,E1 -6360.715,E2 -6360.715} C_VEL
LIN {X 0,Y 495.037,Z 309.814,A -85,B 0,C 180,E1 -6361.394,E2 -6361.394} C_VEL
LIN {X 0,Y 492.162,Z 310.166,A -85,B 0,C 180,E1 -6362.495,E2 -6362.495} C_VEL
LIN {X 0,Y 489.744,Z 310.467,A -85,B 0,C 180,E1 -6363.383,E2 -6363.383} C_VEL
LIN {X 0,Y 488.721,Z 310.604,A -85,B 0,C 180,E1 -6364.07,E2 -6364.07} C_VEL
LIN {X 0,Y 488.646,Z 310.611,A -85,B 0,C 180,E1 -6364.302,E2 -6364.302} C_VEL
LIN {X 0,Y 488.72,Z 310.601,A -85,B 0,C 180,E1 -6367.154,E2 -6367.154} C_VEL
LIN {X 0,Y 488.718,Z 310.607,A -85,B 0,C 180,E1 -6369.811,E2 -6369.811} C_VEL
LIN {X 0,Y 488.681,Z 310.574,A -85,B 0,C 180,E1 -6372.422,E2 -6372.422} C_VEL
LIN {X 0,Y 488.75,Z 310.78,A -85,B 0,C 180,E1 -6374.038,E2 -6374.038} C_VEL
LIN {X 0,Y 488.976,Z 311.795,A -85,B 0,C 180,E1 -6374.173,E2 -6374.173} C_VEL
LIN {X 0,Y 491.82,Z 319.653,A -85,B 0,C 180,E1 -6374.404,E2 -6374.404} C_VEL
LIN {X 0,Y 491.543,Z 391.357,A -85,B 0,C 180,E1 -6375.484,E2 -6375.484} C_VEL
LIN {X 0,Y 491.437,Z 404.435,A -85,B 0,C 180,E1 -6375.851,E2 -6375.851} C_VEL
LIN {X 0,Y 491.258,Z 416.441,A -85,B 0,C 180,E1 -6376.347,E2 -6376.347} C_VEL
LIN {X 0,Y 491.026,Z 428.103,A -85,B 0,C 180,E1 -6376.997,E2 -6376.997} C_VEL
LIN {X 0,Y 490.601,Z 439.296,A -85,B 0,C 180,E1 -6377.802,E2 -6377.802} C_VEL
LIN {X 0,Y 490.216,Z 449.644,A -85,B 0,C 180,E1 -6378.736,E2 -6378.736} C_VEL
LIN {X 0,Y 489.906,Z 458.08,A -85,B 0,C 180,E1 -6379.67,E2 -6379.67} C_VEL
LIN {X 0,Y 489.532,Z 465.847,A -85,B 0,C 180,E1 -6380.706,E2 -6380.706} C_VEL
LIN {X 0,Y 489.24,Z 473.53,A -85,B 0,C 180,E1 -6381.97,E2 -6381.97} C_VEL
LIN {X 0,Y 489.018,Z 479.29,A -85,B 0,C 180,E1 -6383.148,E2 -6383.148} C_VEL
LIN {X 0,Y 488.891,Z 483.571,A -85,B 0,C 180,E1 -6384.225,E2 -6384.225} C_VEL
LIN {X 0,Y 488.665,Z 487.461,A -85,B 0,C 180,E1 -6385.463,E2 -6385.463} C_VEL
LIN {X 0,Y 488.502,Z 490.332,A -85,B 0,C 180,E1 -6386.701,E2 -6386.701} C_VEL
LIN {X 0,Y 488.529,Z 491.697,A -85,B 0,C 180,E1 -6387.527,E2 -6387.527} C_VEL
LIN {X 0,Y 488.42,Z 492.683,A -85,B 0,C 180,E1 -6388.351,E2 -6388.351} C_VEL
LIN {X 0,Y 488.488,Z 493.273,A -85,B 0,C 180,E1 -6389.176,E2 -6389.176} C_VEL
LIN {X 0,Y 488.473,Z 493.506,A -85,B 0,C 180,E1 -6390,E2 -6390} C_VEL
LIN {X 0,Y 488.488,Z 493.324,A -85,B 0,C 180,E1 -6390.824,E2 -6390.824} C_VEL
LIN {X 0,Y 488.42,Z 492.767,A -85,B 0,C 180,E1 -6391.649,E2 -6391.649} C_VEL
LIN {X 0,Y 488.528,Z 491.813,A -85,B 0,C 180,E1 -6392.474,E2 -6392.474} C_VEL
LIN {X 0,Y 488.498,Z 490.501,A -85,B 0,C 180,E1 -6393.299,E2 -6393.299} C_VEL
LIN {X 0,Y 488.661,Z 487.693,A -85,B 0,C 180,E1 -6394.537,E2 -6394.537} C_VEL
LIN {X 0,Y 488.885,Z 483.88,A -85,B 0,C 180,E1 -6395.775,E2 -6395.775} C_VEL
LIN {X 0,Y 488.982,Z 478.796,A -85,B 0,C 180,E1 -6397.061,E2 -6397.061} C_VEL
LIN {X 0,Y 489.335,Z 471.584,A -85,B 0,C 180,E1 -6398.465,E2 -6398.465} C_VEL
LIN {X 0,Y 489.704,Z 463.565,A -85,B 0,C 180,E1 -6399.708,E2 -6399.708} C_VEL
LIN {X 0,Y 490.048,Z 455.343,A -85,B 0,C 180,E1 -6400.745,E2 -6400.745} C_VEL
LIN {X 0,Y 490.376,Z 446.325,A -85,B 0,C 180,E1 -6401.679,E2 -6401.679} C_VEL
LIN {X 0,Y 490.814,Z 435.838,A -85,B 0,C 180,E1 -6402.555,E2 -6402.555} C_VEL
LIN {X 0,Y 491.061,Z 424.351,A -85,B 0,C 180,E1 -6403.323,E2 -6403.323} C_VEL
LIN {X 0,Y 491.31,Z 411.818,A -85,B 0,C 180,E1 -6403.958,E2 -6403.958} C_VEL
LIN {X 0,Y 491.479,Z 399.066,A -85,B 0,C 180,E1 -6404.412,E2 -6404.412} C_VEL
LIN {X 0,Y 491.5,Z 386.301,A -85,B 0,C 180,E1 -6404.703,E2 -6404.703} C_VEL
LIN {X 0,Y 491.803,Z 319.726,A -85,B 0,C 180,E1 -6405.687,E2 -6405.687} C_VEL
LIN {X 0,Y 488.904,Z 311.543,A -85,B 0,C 180,E1 -6405.934,E2 -6405.934} C_VEL
LIN {X 0,Y 488.711,Z 310.685,A -85,B 0,C 180,E1 -6406.097,E2 -6406.097} C_VEL
LIN {X 0,Y 488.713,Z 310.598,A -85,B 0,C 180,E1 -6409.314,E2 -6409.314} C_VEL
LIN {X 0,Y 488.694,Z 310.602,A -85,B 0,C 180,E1 -6411.957,E2 -6411.957} C_VEL
LIN {X 0,Y 488.691,Z 310.611,A -85,B 0,C 180,E1 -6415.038,E2 -6415.038} C_VEL
LIN {X 0,Y 488.69,Z 310.596,A -85,B 0,C 180,E1 -6418.332,E2 -6418.332} C_VEL
LIN {X 0,Y 488.664,Z 310.613,A -85,B 0,C 180,E1 -6421.181,E2 -6421.181} C_VEL
LIN {X 0,Y 488.708,Z 310.606,A -85,B 0,C 180,E1 -6424.114,E2 -6424.114} C_VEL
LIN {X 0,Y 488.656,Z 310.608,A -85,B 0,C 180,E1 -6427.16,E2 -6427.16} C_VEL
LIN {X 0,Y 488.691,Z 310.611,A -85,B 0,C 180,E1 -6430.34,E2 -6430.34} C_VEL
LIN {X 0,Y 488.661,Z 310.602,A -85,B 0,C 180,E1 -6433.656,E2 -6433.656} C_VEL
LIN {X 0,Y 488.66,Z 310.615,A -85,B 0,C 180,E1 -6436.342,E2 -6436.342} C_VEL
LIN {X 0,Y 488.699,Z 310.599,A -85,B 0,C 180,E1 -6439.673,E2 -6439.673} C_VEL
LIN {X 0,Y 488.659,Z 310.614,A -85,B 0,C 180,E1 -6442.839,E2 -6442.839} C_VEL
LIN {X 0,Y 488.711,Z 310.606,A -85,B 0,C 180,E1 -6445.885,E2 -6445.885} C_VEL
LIN {X 0,Y 488.675,Z 310.599,A -85,B 0,C 180,E1 -6448.819,E2 -6448.819} C_VEL
LIN {X 0,Y 488.686,Z 310.593,A -85,B 0,C 180,E1 -6451.667,E2 -6451.667} C_VEL
LIN {X 0,Y 488.683,Z 310.611,A -85,B 0,C 180,E1 -6454.441,E2 -6454.441} C_VEL
LIN {X 0,Y 488.699,Z 310.606,A -85,B 0,C 180,E1 -6457.152,E2 -6457.152} C_VEL
LIN {X 0,Y 488.704,Z 310.601,A -85,B 0,C 180,E1 -6459.809,E2 -6459.809} C_VEL
LIN {X 0,Y 488.681,Z 310.616,A -85,B 0,C 180,E1 -6462.421,E2 -6462.421} C_VEL
LIN {X 0,Y 488.743,Z 310.595,A -85,B 0,C 180,E1 -6464.999,E2 -6464.999} C_VEL
LIN {X 0,Y 488.795,Z 310.601,A -85,B 0,C 180,E1 -6468.387,E2 -6468.387} C_VEL
LIN {X 0,Y 488.75,Z 310.596,A -85,B 0,C 180,E1 -6471.732,E2 -6471.732} C_VEL
LIN {X 0,Y 488.794,Z 310.597,A -85,B 0,C 180,E1 -6474.223,E2 -6474.223} C_VEL
LIN {X 0,Y 488.939,Z 310.574,A -85,B 0,C 180,E1 -6477.528,E2 -6477.528} C_VEL
LIN {X 0,Y 488.884,Z 310.584,A -85,B 0,C 180,E1 -6480.824,E2 -6480.824} C_VEL
LIN {X 0,Y 488.931,Z 310.583,A -85,B 0,C 180,E1 -6482.471,E2 -6482.471} C_VEL
LIN {X 0,Y 488.825,Z 310.587,A -85,B 0,C 180,E1 -6485.776,E2 -6485.776} C_VEL
LIN {X 0,Y 488.765,Z 310.603,A -85,B 0,C 180,E1 -6488.267,E2 -6488.267} C_VEL
LIN {X 0,Y 488.775,Z 310.595,A -85,B 0,C 180,E1 -6491.613,E2 -6491.613} C_VEL
LIN {X 0,Y 488.752,Z 310.6,A -85,B 0,C 180,E1 -6495.001,E2 -6495.001} C_VEL
LIN {X 0,Y 488.736,Z 310.6,A -85,B 0,C 180,E1 -6498.443,E2 -6498.443} C_VEL
LIN {X 0,Y 488.699,Z 310.596,A -85,B 0,C 180,E1 -6501.071,E2 -6501.071} C_VEL
LIN {X 0,Y 488.662,Z 310.612,A -85,B 0,C 180,E1 -6503.747,E2 -6503.747} C_VEL
LIN {X 0,Y 488.691,Z 310.603,A -85,B 0,C 180,E1 -6506.922,E2 -6506.922} C_VEL
LIN {X 0,Y 488.716,Z 310.609,A -85,B 0,C 180,E1 -6510.22,E2 -6510.22} C_VEL
LIN {X 0,Y 488.704,Z 310.605,A -85,B 0,C 180,E1 -6513.48,E2 -6513.48} C_VEL
LIN {X 0,Y 488.643,Z 310.619,A -85,B 0,C 180,E1 -6516.35,E2 -6516.35} C_VEL
LIN {X 0,Y 488.682,Z 310.605,A -85,B 0,C 180,E1 -6519.256,E2 -6519.256} C_VEL
LIN {X 0,Y 488.662,Z 310.611,A -85,B 0,C 180,E1 -6522.529,E2 -6522.529} C_VEL
LIN {X 0,Y 488.693,Z 310.592,A -85,B 0,C 180,E1 -6525.197,E2 -6525.197} C_VEL
LIN {X 0,Y 488.658,Z 310.612,A -85,B 0,C 180,E1 -6528.58,E2 -6528.58} C_VEL
LIN {X 0,Y 488.685,Z 310.604,A -85,B 0,C 180,E1 -6530.95,E2 -6530.95} C_VEL
LIN {X 0,Y 488.643,Z 310.614,A -85,B 0,C 180,E1 -6533.866,E2 -6533.866} C_VEL
LIN {X 0,Y 488.708,Z 310.605,A -85,B 0,C 180,E1 -6536.521,E2 -6536.521} C_VEL
LIN {X 0,Y 488.704,Z 310.59,A -85,B 0,C 180,E1 -6539.78,E2 -6539.78} C_VEL
LIN {X 0,Y 488.813,Z 310.85,A -85,B 0,C 180,E1 -6540.544,E2 -6540.544} C_VEL
LIN {X 0,Y 491.797,Z 324.991,A -85,B 0,C 180,E1 -6542.583,E2 -6542.583} C_VEL
LIN {X 0,Y 491.305,Z 344.055,A -85,B 0,C 180,E1 -6545.04,E2 -6545.04} C_VEL
LIN {X 0,Y 490.417,Z 371.148,A -85,B 0,C 180,E1 -6548.462,E2 -6548.462} C_VEL
LIN {X 0,Y 489.712,Z 397.851,A -85,B 0,C 180,E1 -6551.812,E2 -6551.812} C_VEL
LIN {X 0,Y 489.324,Z 413.033,A -85,B 0,C 180,E1 -6553.693,E2 -6553.693} C_VEL
LIN {X 0,Y 491.525,Z 434.212,A -85,B 0,C 180,E1 -6554.094,E2 -6554.094} C_VEL
LIN {X 0,Y 490.98,Z 523.362,A -85,B 0,C 180,E1 -6555.414,E2 -6555.414} C_VEL
LIN {X 0,Y 490.626,Z 536.708,A -85,B 0,C 180,E1 -6555.774,E2 -6555.774} C_VEL
LIN {X 0,Y 490.262,Z 548.97,A -85,B 0,C 180,E1 -6556.266,E2 -6556.266} C_VEL
LIN {X 0,Y 489.809,Z 559.831,A -85,B 0,C 180,E1 -6556.844,E2 -6556.844} C_VEL
LIN {X 0,Y 489.437,Z 570.469,A -85,B 0,C 180,E1 -6557.562,E2 -6557.562} C_VEL
LIN {X 0,Y 489.039,Z 581.545,A -85,B 0,C 180,E1 -6558.498,E2 -6558.498} C_VEL
LIN {X 0,Y 488.747,Z 590.6,A -85,B 0,C 180,E1 -6559.436,E2 -6559.436} C_VEL
LIN {X 0,Y 488.439,Z 600.457,A -85,B 0,C 180,E1 -6560.685,E2 -6560.685} C_VEL
LIN {X 0,Y 488.275,Z 608.336,A -85,B 0,C 180,E1 -6561.933,E2 -6561.933} C_VEL
LIN {X 0,Y 488.182,Z 615.613,A -85,B 0,C 180,E1 -6563.387,E2 -6563.387} C_VEL
LIN {X 0,Y 488.144,Z 620.464,A -85,B 0,C 180,E1 -6564.63,E2 -6564.63} C_VEL
LIN {X 0,Y 488.232,Z 624.19,A -85,B 0,C 180,E1 -6565.873,E2 -6565.873} C_VEL
LIN {X 0,Y 488.169,Z 626.098,A -85,B 0,C 180,E1 -6566.699,E2 -6566.699} C_VEL
LIN {X 0,Y 488.136,Z 627.531,A -85,B 0,C 180,E1 -6567.524,E2 -6567.524} C_VEL
LIN {X 0,Y 488.196,Z 629.191,A -85,B 0,C 180,E1 -6569.175,E2 -6569.175} C_VEL
LIN {X 0,Y 488.186,Z 629.413,A -85,B 0,C 180,E1 -6570,E2 -6570} C_VEL
LIN {X 0,Y 488.196,Z 629.192,A -85,B 0,C 180,E1 -6570.825,E2 -6570.825} C_VEL
LIN {X 0,Y 488.136,Z 627.535,A -85,B 0,C 180,E1 -6572.475,E2 -6572.475} C_VEL
LIN {X 0,Y 488.168,Z 626.102,A -85,B 0,C 180,E1 -6573.301,E2 -6573.301} C_VEL
LIN {X 0,Y 488.161,Z 623.081,A -85,B 0,C 180,E1 -6574.542,E2 -6574.542} C_VEL
LIN {X 0,Y 488.22,Z 617.883,A -85,B 0,C 180,E1 -6576.069,E2 -6576.069} C_VEL
LIN {X 0,Y 488.235,Z 611.685,A -85,B 0,C 180,E1 -6577.444,E2 -6577.444} C_VEL
LIN {X 0,Y 488.34,Z 604.616,A -85,B 0,C 180,E1 -6578.691,E2 -6578.691} C_VEL
LIN {X 0,Y 488.563,Z 595.795,A -85,B 0,C 180,E1 -6579.94,E2 -6579.94} C_VEL
LIN {X 0,Y 488.872,Z 585.783,A -85,B 0,C 180,E1 -6581.086,E2 -6581.086} C_VEL
LIN {X 0,Y 489.336,Z 576.083,A -85,B 0,C 180,E1 -6581.989,E2 -6581.989} C_VEL
LIN {X 0,Y 489.614,Z 566.293,A -85,B 0,C 180,E1 -6582.739,E2 -6582.739} C_VEL
LIN {X 0,Y 490.001,Z 554.135,A -85,B 0,C 180,E1 -6583.478,E2 -6583.478} C_VEL
LIN {X 0,Y 490.48,Z 541.698,A -85,B 0,C 180,E1 -6584.045,E2 -6584.045} C_VEL
LIN {X 0,Y 490.842,Z 528.957,A -85,B 0,C 180,E1 -6584.458,E2 -6584.458} C_VEL
LIN {X 0,Y 491.086,Z 515.689,A -85,B 0,C 180,E1 -6584.715,E2 -6584.715} C_VEL
LIN {X 0,Y 491.39,Z 431.975,A -85,B 0,C 180,E1 -6585.944,E2 -6585.944} C_VEL
LIN {X 0,Y 489.339,Z 413.031,A -85,B 0,C 180,E1 -6586.307,E2 -6586.307} C_VEL
LIN {X 0,Y 489.909,Z 389.255,A -85,B 0,C 180,E1 -6589.265,E2 -6589.265} C_VEL
LIN {X 0,Y 490.633,Z 364.997,A -85,B 0,C 180,E1 -6592.308,E2 -6592.308} C_VEL
LIN {X 0,Y 491.448,Z 339.023,A -85,B 0,C 180,E1 -6595.6,E2 -6595.6} C_VEL
LIN {X 0,Y 491.798,Z 324.975,A -85,B 0,C 180,E1 -6597.417,E2 -6597.417} C_VEL
LIN {X 0,Y 488.768,Z 310.708,A -85,B 0,C 180,E1 -6599.503,E2 -6599.503} C_VEL
LIN {X 0,Y 488.699,Z 310.605,A -85,B 0,C 180,E1 -6603.125,E2 -6603.125} C_VEL
LIN {X 0,Y 488.704,Z 310.607,A -85,B 0,C 180,E1 -6605.115,E2 -6605.115} C_VEL
LIN {X 0,Y 488.653,Z 310.614,A -85,B 0,C 180,E1 -6608.202,E2 -6608.202} C_VEL
LIN {X 0,Y 488.69,Z 310.609,A -85,B 0,C 180,E1 -6610.34,E2 -6610.34} C_VEL
LIN {X 0,Y 488.668,Z 310.611,A -85,B 0,C 180,E1 -6613.655,E2 -6613.655} C_VEL
LIN {X 0,Y 488.67,Z 310.611,A -85,B 0,C 180,E1 -6616.344,E2 -6616.344} C_VEL
LIN {X 0,Y 488.698,Z 310.612,A -85,B 0,C 180,E1 -6619.673,E2 -6619.673} C_VEL
LIN {X 0,Y 488.643,Z 310.587,A -85,B 0,C 180,E1 -6622.838,E2 -6622.838} C_VEL
LIN {X 0,Y 488.71,Z 310.603,A -85,B 0,C 180,E1 -6625.885,E2 -6625.885} C_VEL
LIN {X 0,Y 488.685,Z 310.608,A -85,B 0,C 180,E1 -6628.82,E2 -6628.82} C_VEL
LIN {X 0,Y 488.704,Z 310.603,A -85,B 0,C 180,E1 -6631.669,E2 -6631.669} C_VEL
LIN {X 0,Y 488.691,Z 310.607,A -85,B 0,C 180,E1 -6634.959,E2 -6634.959} C_VEL
LIN {X 0,Y 488.689,Z 310.602,A -85,B 0,C 180,E1 -6638.043,E2 -6638.043} C_VEL
LIN {X 0,Y 488.731,Z 310.596,A -85,B 0,C 180,E1 -6640.686,E2 -6640.686} C_VEL
LIN {X 0,Y 488.752,Z 310.603,A -85,B 0,C 180,E1 -6644.145,E2 -6644.145} C_VEL
LIN {X 0,Y 488.73,Z 310.601,A -85,B 0,C 180,E1 -6647.543,E2 -6647.543} C_VEL
LIN {X 0,Y 488.744,Z 310.605,A -85,B 0,C 180,E1 -6650.064,E2 -6650.064} C_VEL
LIN {X 0,Y 488.852,Z 310.583,A -85,B 0,C 180,E1 -6652.731,E2 -6652.731} C_VEL
LIN {X 0,Y 488.791,Z 310.591,A -85,B 0,C 180,E1 -6655.051,E2 -6655.051} C_VEL
LIN {X 0,Y 488.932,Z 310.583,A -85,B 0,C 180,E1 -6657.529,E2 -6657.529} C_VEL
LIN {X 0,Y 488.93,Z 310.574,A -85,B 0,C 180,E1 -6660,E2 -6660} C_VEL
LIN {X 0,Y 488.94,Z 310.574,A -85,B 0,C 180,E1 -6662.472,E2 -6662.472} C_VEL
LIN {X 0,Y 488.806,Z 310.596,A -85,B 0,C 180,E1 -6665.776,E2 -6665.776} C_VEL
LIN {X 0,Y 488.77,Z 310.593,A -85,B 0,C 180,E1 -6668.267,E2 -6668.267} C_VEL
LIN {X 0,Y 488.796,Z 310.601,A -85,B 0,C 180,E1 -6671.613,E2 -6671.613} C_VEL
LIN {X 0,Y 488.745,Z 310.594,A -85,B 0,C 180,E1 -6675.001,E2 -6675.001} C_VEL
LIN {X 0,Y 488.736,Z 310.601,A -85,B 0,C 180,E1 -6678.443,E2 -6678.443} C_VEL
LIN {X 0,Y 488.699,Z 310.603,A -85,B 0,C 180,E1 -6681.071,E2 -6681.071} C_VEL
LIN {X 0,Y 488.661,Z 310.617,A -85,B 0,C 180,E1 -6683.747,E2 -6683.747} C_VEL
LIN {X 0,Y 488.691,Z 310.604,A -85,B 0,C 180,E1 -6686.922,E2 -6686.922} C_VEL
LIN {X 0,Y 488.701,Z 310.591,A -85,B 0,C 180,E1 -6690.221,E2 -6690.221} C_VEL
LIN {X 0,Y 488.704,Z 310.61,A -85,B 0,C 180,E1 -6693.48,E2 -6693.48} C_VEL
LIN {X 0,Y 488.667,Z 310.608,A -85,B 0,C 180,E1 -6696.353,E2 -6696.353} C_VEL
LIN {X 0,Y 488.682,Z 310.599,A -85,B 0,C 180,E1 -6699.256,E2 -6699.256} C_VEL
LIN {X 0,Y 488.662,Z 310.615,A -85,B 0,C 180,E1 -6701.595,E2 -6701.595} C_VEL
LIN {X 0,Y 488.695,Z 310.607,A -85,B 0,C 180,E1 -6704.804,E2 -6704.804} C_VEL
LIN {X 0,Y 488.644,Z 310.61,A -85,B 0,C 180,E1 -6707.47,E2 -6707.47} C_VEL
LIN {X 0,Y 488.701,Z 310.611,A -85,B 0,C 180,E1 -6709.674,E2 -6709.674} C_VEL
LIN {X 0,Y 488.658,Z 310.607,A -85,B 0,C 180,E1 -6712.84,E2 -6712.84} C_VEL
LIN {X 0,Y 488.715,Z 310.605,A -85,B 0,C 180,E1 -6715.887,E2 -6715.887} C_VEL
LIN {X 0,Y 488.665,Z 310.612,A -85,B 0,C 180,E1 -6718.819,E2 -6718.819} C_VEL
LIN {X 0,Y 488.691,Z 310.597,A -85,B 0,C 180,E1 -6721.668,E2 -6721.668} C_VEL
LIN {X 0,Y 488.646,Z 310.611,A -85,B 0,C 180,E1 -6724.302,E2 -6724.302} C_VEL
LIN {X 0,Y 488.005,Z 310.699,A -85,B 0,C 180,E1 -6724.99,E2 -6724.99} C_VEL
LIN {X 0,Y 485.177,Z 311.047,A -85,B 0,C 180,E1 -6726.108,E2 -6726.108} C_VEL
LIN {X 0,Y 482.766,Z 311.344,A -85,B 0,C 180,E1 -6727.009,E2 -6727.009} C_VEL
LIN {X 0,Y 481.723,Z 311.468,A -85,B 0,C 180,E1 -6727.704,E2 -6727.704} C_VEL
LIN {X 0,Y 481.635,Z 311.479,A -85,B 0,C 180,E1 -6727.94,E2 -6727.94} C_VEL
LIN {X 0,Y 481.694,Z 311.481,A -85,B 0,C 180,E1 -6730.393,E2 -6730.393} C_VEL
LIN {X 0,Y 481.697,Z 311.595,A -85,B 0,C 180,E1 -6733.77,E2 -6733.77} C_VEL
LIN {X 0,Y 481.916,Z 312.548,A -85,B 0,C 180,E1 -6733.928,E2 -6733.928} C_VEL
LIN {X 0,Y 484.995,Z 320.962,A -85,B 0,C 180,E1 -6734.183,E2 -6734.183} C_VEL
LIN {X 0,Y 484.74,Z 392.354,A -85,B 0,C 180,E1 -6735.275,E2 -6735.275} C_VEL
LIN {X 0,Y 484.615,Z 405.427,A -85,B 0,C 180,E1 -6735.647,E2 -6735.647} C_VEL
LIN {X 0,Y 484.439,Z 417.427,A -85,B 0,C 180,E1 -6736.151,E2 -6736.151} C_VEL
LIN {X 0,Y 484.185,Z 428.69,A -85,B 0,C 180,E1 -6736.784,E2 -6736.784} C_VEL
LIN {X 0,Y 483.731,Z 440.28,A -85,B 0,C 180,E1 -6737.626,E2 -6737.626} C_VEL
LIN {X 0,Y 483.324,Z 450.627,A -85,B 0,C 180,E1 -6738.573,E2 -6738.573} C_VEL
LIN {X 0,Y 482.994,Z 459.062,A -85,B 0,C 180,E1 -6739.521,E2 -6739.521} C_VEL
LIN {X 0,Y 482.599,Z 466.828,A -85,B 0,C 180,E1 -6740.571,E2 -6740.571} C_VEL
LIN {X 0,Y 482.282,Z 474.51,A -85,B 0,C 180,E1 -6741.853,E2 -6741.853} C_VEL
LIN {X 0,Y 482.041,Z 480.27,A -85,B 0,C 180,E1 -6743.049,E2 -6743.049} C_VEL
LIN {X 0,Y 481.906,Z 484.549,A -85,B 0,C 180,E1 -6744.141,E2 -6744.141} C_VEL
LIN {X 0,Y 481.655,Z 488.441,A -85,B 0,C 180,E1 -6745.397,E2 -6745.397} C_VEL
LIN {X 0,Y 481.482,Z 491.312,A -85,B 0,C 180,E1 -6746.653,E2 -6746.653} C_VEL
LIN {X 0,Y 481.514,Z 492.675,A -85,B 0,C 180,E1 -6747.49,E2 -6747.49} C_VEL
LIN {X 0,Y 481.399,Z 493.661,A -85,B 0,C 180,E1 -6748.327,E2 -6748.327} C_VEL
LIN {X 0,Y 481.47,Z 494.25,A -85,B 0,C 180,E1 -6749.164,E2 -6749.164} C_VEL
LIN {X 0,Y 481.455,Z 494.483,A -85,B 0,C 180,E1 -6750,E2 -6750} C_VEL
LIN {X 0,Y 481.47,Z 494.3,A -85,B 0,C 180,E1 -6750.836,E2 -6750.836} C_VEL
LIN {X 0,Y 481.399,Z 493.743,A -85,B 0,C 180,E1 -6751.673,E2 -6751.673} C_VEL
LIN {X 0,Y 481.513,Z 492.79,A -85,B 0,C 180,E1 -6752.51,E2 -6752.51} C_VEL
LIN {X 0,Y 481.477,Z 491.479,A -85,B 0,C 180,E1 -6753.347,E2 -6753.347} C_VEL
LIN {X 0,Y 481.651,Z 488.67,A -85,B 0,C 180,E1 -6754.603,E2 -6754.603} C_VEL
LIN {X 0,Y 481.899,Z 484.856,A -85,B 0,C 180,E1 -6755.859,E2 -6755.859} C_VEL
LIN {X 0,Y 482.007,Z 479.774,A -85,B 0,C 180,E1 -6757.163,E2 -6757.163} C_VEL
LIN {X 0,Y 482.386,Z 472.559,A -85,B 0,C 180,E1 -6758.588,E2 -6758.588} C_VEL
LIN {X 0,Y 482.782,Z 464.539,A -85,B 0,C 180,E1 -6759.849,E2 -6759.849} C_VEL
LIN {X 0,Y 483.144,Z 456.318,A -85,B 0,C 180,E1 -6760.9,E2 -6760.9} C_VEL
LIN {X 0,Y 483.494,Z 447.298,A -85,B 0,C 180,E1 -6761.848,E2 -6761.848} C_VEL
LIN {X 0,Y 483.956,Z 436.81,A -85,B 0,C 180,E1 -6762.736,E2 -6762.736} C_VEL
LIN {X 0,Y 484.225,Z 425.322,A -85,B 0,C 180,E1 -6763.514,E2 -6763.514} C_VEL
LIN {X 0,Y 484.487,Z 412.786,A -85,B 0,C 180,E1 -6764.158,E2 -6764.158} C_VEL
LIN {X 0,Y 484.658,Z 400.031,A -85,B 0,C 180,E1 -6764.62,E2 -6764.62} C_VEL
LIN {X 0,Y 484.68,Z 387.258,A -85,B 0,C 180,E1 -6764.914,E2 -6764.914} C_VEL
LIN {X 0,Y 484.996,Z 321.111,A -85,B 0,C 180,E1 -6765.907,E2 -6765.907} C_VEL
LIN {X 0,Y 481.878,Z 312.512,A -85,B 0,C 180,E1 -6766.168,E2 -6766.168} C_VEL
LIN {X 0,Y 481.687,Z 311.6,A -85,B 0,C 180,E1 -6766.319,E2 -6766.319} C_VEL
LIN {X 0,Y 481.652,Z 311.458,A -85,B 0,C 180,E1 -6768.724,E2 -6768.724} C_VEL
LIN {X 0,Y 481.641,Z 311.483,A -85,B 0,C 180,E1 -6771.395,E2 -6771.395} C_VEL
LIN {X 0,Y 481.641,Z 311.486,A -85,B 0,C 180,E1 -6774.115,E2 -6774.115} C_VEL
LIN {X 0,Y 481.641,Z 311.471,A -85,B 0,C 180,E1 -6777.114,E2 -6777.114} C_VEL
LIN {X 0,Y 481.65,Z 311.484,A -85,B 0,C 180,E1 -6779.742,E2 -6779.742} C_VEL
LIN {X 0,Y 481.632,Z 311.487,A -85,B 0,C 180,E1 -6782.677,E2 -6782.677} C_VEL
LIN {X 0,Y 481.623,Z 311.488,A -85,B 0,C 180,E1 -6785.71,E2 -6785.71} C_VEL
LIN {X 0,Y 481.652,Z 311.489,A -85,B 0,C 180,E1 -6788.86,E2 -6788.86} C_VEL
LIN {X 0,Y 481.617,Z 311.486,A -85,B 0,C 180,E1 -6791.908,E2 -6791.908} C_VEL
LIN {X 0,Y 481.646,Z 311.481,A -85,B 0,C 180,E1 -6794.458,E2 -6794.458} C_VEL
LIN {X 0,Y 481.607,Z 311.495,A -85,B 0,C 180,E1 -6796.855,E2 -6796.855} C_VEL
LIN {X 0,Y 481.65,Z 311.478,A -85,B 0,C 180,E1 -6800.057,E2 -6800.057} C_VEL
LIN {X 0,Y 481.613,Z 311.487,A -85,B 0,C 180,E1 -6803.377,E2 -6803.377} C_VEL
LIN {X 0,Y 481.665,Z 311.488,A -85,B 0,C 180,E1 -6806.326,E2 -6806.326} C_VEL
LIN {X 0,Y 481.626,Z 311.471,A -85,B 0,C 180,E1 -6809.421,E2 -6809.421} C_VEL
LIN {X 0,Y 481.642,Z 311.473,A -85,B 0,C 180,E1 -6812.164,E2 -6812.164} C_VEL
LIN {X 0,Y 481.666,Z 311.485,A -85,B 0,C 180,E1 -6814.967,E2 -6814.967} C_VEL
LIN {X 0,Y 481.628,Z 311.486,A -85,B 0,C 180,E1 -6817.704,E2 -6817.704} C_VEL
LIN {X 0,Y 481.683,Z 311.482,A -85,B 0,C 180,E1 -6820.392,E2 -6820.392} C_VEL
LIN {X 0,Y 481.643,Z 311.485,A -85,B 0,C 180,E1 -6823.032,E2 -6823.032} C_VEL
LIN {X 0,Y 481.663,Z 311.475,A -85,B 0,C 180,E1 -6825.638,E2 -6825.638} C_VEL
LIN {X 0,Y 481.741,Z 311.477,A -85,B 0,C 180,E1 -6828.215,E2 -6828.215} C_VEL
LIN {X 0,Y 481.709,Z 311.472,A -85,B 0,C 180,E1 -6831.611,E2 -6831.611} C_VEL
LIN {X 0,Y 481.756,Z 311.473,A -85,B 0,C 180,E1 -6834.139,E2 -6834.139} C_VEL
LIN {X 0,Y 481.906,Z 311.45,A -85,B 0,C 180,E1 -6837.492,E2 -6837.492} C_VEL
LIN {X 0,Y 481.837,Z 311.462,A -85,B 0,C 180,E1 -6840.836,E2 -6840.836} C_VEL
LIN {X 0,Y 481.897,Z 311.459,A -85,B 0,C 180,E1 -6842.508,E2 -6842.508} C_VEL
LIN {X 0,Y 481.785,Z 311.465,A -85,B 0,C 180,E1 -6845.861,E2 -6845.861} C_VEL
LIN {X 0,Y 481.719,Z 311.482,A -85,B 0,C 180,E1 -6848.389,E2 -6848.389} C_VEL
LIN {X 0,Y 481.726,Z 311.475,A -85,B 0,C 180,E1 -6851.786,E2 -6851.786} C_VEL
LIN {X 0,Y 481.734,Z 311.473,A -85,B 0,C 180,E1 -6855.225,E2 -6855.225} C_VEL
LIN {X 0,Y 481.698,Z 311.473,A -85,B 0,C 180,E1 -6858.722,E2 -6858.722} C_VEL
LIN {X 0,Y 481.637,Z 311.475,A -85,B 0,C 180,E1 -6861.395,E2 -6861.395} C_VEL
LIN {X 0,Y 481.641,Z 311.491,A -85,B 0,C 180,E1 -6864.115,E2 -6864.115} C_VEL
LIN {X 0,Y 481.665,Z 311.478,A -85,B 0,C 180,E1 -6867.122,E2 -6867.122} C_VEL
LIN {X 0,Y 481.665,Z 311.479,A -85,B 0,C 180,E1 -6869.742,E2 -6869.742} C_VEL
LIN {X 0,Y 481.646,Z 311.485,A -85,B 0,C 180,E1 -6872.676,E2 -6872.676} C_VEL
LIN {X 0,Y 481.643,Z 311.481,A -85,B 0,C 180,E1 -6875.202,E2 -6875.202} C_VEL
LIN {X 0,Y 481.625,Z 311.494,A -85,B 0,C 180,E1 -6878.004,E2 -6878.004} C_VEL
LIN {X 0,Y 481.621,Z 311.488,A -85,B 0,C 180,E1 -6881.046,E2 -6881.046} C_VEL
LIN {X 0,Y 481.649,Z 311.471,A -85,B 0,C 180,E1 -6884.459,E2 -6884.459} C_VEL
LIN {X 0,Y 481.61,Z 311.495,A -85,B 0,C 180,E1 -6887.836,E2 -6887.836} C_VEL
LIN {X 0,Y 481.645,Z 311.481,A -85,B 0,C 180,E1 -6890.657,E2 -6890.657} C_VEL
LIN {X 0,Y 481.604,Z 311.493,A -85,B 0,C 180,E1 -6893.38,E2 -6893.38} C_VEL
LIN {X 0,Y 481.668,Z 311.484,A -85,B 0,C 180,E1 -6896.327,E2 -6896.327} C_VEL
LIN {X 0,Y 481.658,Z 311.466,A -85,B 0,C 180,E1 -6899.775,E2 -6899.775} C_VEL
LIN {X 0,Y 481.723,Z 311.756,A -85,B 0,C 180,E1 -6900.313,E2 -6900.313} C_VEL
LIN {X 0,Y 484.772,Z 325.662,A -85,B 0,C 180,E1 -6902.36,E2 -6902.36} C_VEL
LIN {X 0,Y 484.883,Z 330.937,A -85,B 0,C 180,E1 -6903.068,E2 -6903.068} C_VEL
LIN {X 0,Y 484.021,Z 354.868,A -85,B 0,C 180,E1 -6906.172,E2 -6906.172} C_VEL
LIN {X 0,Y 483.242,Z 377.975,A -85,B 0,C 180,E1 -6909.126,E2 -6909.126} C_VEL
LIN {X 0,Y 482.528,Z 403.709,A -85,B 0,C 180,E1 -6912.409,E2 -6912.409} C_VEL
LIN {X 0,Y 482.309,Z 412.043,A -85,B 0,C 180,E1 -6913.449,E2 -6913.449} C_VEL
LIN {X 0,Y 484.667,Z 434.982,A -85,B 0,C 180,E1 -6913.889,E2 -6913.889} C_VEL
LIN {X 0,Y 484.105,Z 522.38,A -85,B 0,C 180,E1 -6915.202,E2 -6915.202} C_VEL
LIN {X 0,Y 483.737,Z 535.723,A -85,B 0,C 180,E1 -6915.567,E2 -6915.567} C_VEL
LIN {X 0,Y 483.302,Z 547.976,A -85,B 0,C 180,E1 -6916.064,E2 -6916.064} C_VEL
LIN {X 0,Y 482.779,Z 560.372,A -85,B 0,C 180,E1 -6916.746,E2 -6916.746} C_VEL
LIN {X 0,Y 482.353,Z 572.517,A -85,B 0,C 180,E1 -6917.622,E2 -6917.622} C_VEL
LIN {X 0,Y 481.922,Z 583.795,A -85,B 0,C 180,E1 -6918.646,E2 -6918.646} C_VEL
LIN {X 0,Y 481.566,Z 593.134,A -85,B 0,C 180,E1 -6919.702,E2 -6919.702} C_VEL
LIN {X 0,Y 481.312,Z 602.264,A -85,B 0,C 180,E1 -6920.969,E2 -6920.969} C_VEL
LIN {X 0,Y 481.178,Z 609.636,A -85,B 0,C 180,E1 -6922.236,E2 -6922.236} C_VEL
LIN {X 0,Y 481.12,Z 616.131,A -85,B 0,C 180,E1 -6923.65,E2 -6923.65} C_VEL
LIN {X 0,Y 481.096,Z 620.831,A -85,B 0,C 180,E1 -6924.972,E2 -6924.972} C_VEL
LIN {X 0,Y 481.157,Z 623.203,A -85,B 0,C 180,E1 -6925.812,E2 -6925.812} C_VEL
LIN {X 0,Y 481.121,Z 625.115,A -85,B 0,C 180,E1 -6926.65,E2 -6926.65} C_VEL
LIN {X 0,Y 481.093,Z 626.55,A -85,B 0,C 180,E1 -6927.488,E2 -6927.488} C_VEL
LIN {X 0,Y 481.176,Z 628.214,A -85,B 0,C 180,E1 -6929.163,E2 -6929.163} C_VEL
LIN {X 0,Y 481.166,Z 628.436,A -85,B 0,C 180,E1 -6930,E2 -6930} C_VEL
LIN {X 0,Y 481.176,Z 628.215,A -85,B 0,C 180,E1 -6930.837,E2 -6930.837} C_VEL
LIN {X 0,Y 481.093,Z 626.554,A -85,B 0,C 180,E1 -6932.512,E2 -6932.512} C_VEL
LIN {X 0,Y 481.121,Z 625.119,A -85,B 0,C 180,E1 -6933.35,E2 -6933.35} C_VEL
LIN {X 0,Y 481.107,Z 622.096,A -85,B 0,C 180,E1 -6934.608,E2 -6934.608} C_VEL
LIN {X 0,Y 481.13,Z 618.011,A -85,B 0,C 180,E1 -6935.869,E2 -6935.869} C_VEL
LIN {X 0,Y 481.152,Z 611.73,A -85,B 0,C 180,E1 -6937.343,E2 -6937.343} C_VEL
LIN {X 0,Y 481.267,Z 604.889,A -85,B 0,C 180,E1 -6938.608,E2 -6938.608} C_VEL
LIN {X 0,Y 481.449,Z 596.42,A -85,B 0,C 180,E1 -6939.876,E2 -6939.876} C_VEL
LIN {X 0,Y 481.778,Z 587.77,A -85,B 0,C 180,E1 -6940.932,E2 -6940.932} C_VEL
LIN {X 0,Y 482.105,Z 579.465,A -85,B 0,C 180,E1 -6941.776,E2 -6941.776} C_VEL
LIN {X 0,Y 482.526,Z 568.037,A -85,B 0,C 180,E1 -6942.726,E2 -6942.726} C_VEL
LIN {X 0,Y 482.88,Z 556.867,A -85,B 0,C 180,E1 -6943.466,E2 -6943.466} C_VEL
LIN {X 0,Y 483.414,Z 544.544,A -85,B 0,C 180,E1 -6944.094,E2 -6944.094} C_VEL
LIN {X 0,Y 483.828,Z 531.635,A -85,B 0,C 180,E1 -6944.565,E2 -6944.565} C_VEL
LIN {X 0,Y 484.188,Z 517.996,A -85,B 0,C 180,E1 -6944.876,E2 -6944.876} C_VEL
LIN {X 0,Y 484.536,Z 432.455,A -85,B 0,C 180,E1 -6946.153,E2 -6946.153} C_VEL
LIN {X 0,Y 482.316,Z 411.886,A -85,B 0,C 180,E1 -6946.562,E2 -6946.562} C_VEL
LIN {X 0,Y 482.992,Z 386.582,A -85,B 0,C 180,E1 -6949.774,E2 -6949.774} C_VEL
LIN {X 0,Y 483.69,Z 364.078,A -85,B 0,C 180,E1 -6952.646,E2 -6952.646} C_VEL
LIN {X 0,Y 484.496,Z 341.392,A -85,B 0,C 180,E1 -6955.565,E2 -6955.565} C_VEL
LIN {X 0,Y 484.975,Z 327.419,A -85,B 0,C 180,E1 -6957.393,E2 -6957.393} C_VEL
LIN {X 0,Y 482.618,Z 315.57,A -85,B 0,C 180,E1 -6959.104,E2 -6959.104} C_VEL
LIN {X 0,Y 481.701,Z 311.585,A -85,B 0,C 180,E1 -6959.739,E2 -6959.739} C_VEL
LIN {X 0,Y 481.649,Z 311.483,A -85,B 0,C 180,E1 -6962.675,E2 -6962.675} C_VEL
LIN {X 0,Y 481.647,Z 311.486,A -85,B 0,C 180,E1 -6965.201,E2 -6965.201} C_VEL
LIN {X 0,Y 481.628,Z 311.492,A -85,B 0,C 180,E1 -6968.003,E2 -6968.003} C_VEL
LIN {X 0,Y 481.619,Z 311.488,A -85,B 0,C 180,E1 -6971.045,E2 -6971.045} C_VEL
LIN {X 0,Y 481.649,Z 311.471,A -85,B 0,C 180,E1 -6974.458,E2 -6974.458} C_VEL
LIN {X 0,Y 481.62,Z 311.493,A -85,B 0,C 180,E1 -6977.836,E2 -6977.836} C_VEL
LIN {X 0,Y 481.643,Z 311.478,A -85,B 0,C 180,E1 -6980.655,E2 -6980.655} C_VEL
LIN {X 0,Y 481.602,Z 311.465,A -85,B 0,C 180,E1 -6983.379,E2 -6983.379} C_VEL
LIN {X 0,Y 481.664,Z 311.484,A -85,B 0,C 180,E1 -6986.326,E2 -6986.326} C_VEL
LIN {X 0,Y 481.644,Z 311.488,A -85,B 0,C 180,E1 -6989.417,E2 -6989.417} C_VEL
LIN {X 0,Y 481.654,Z 311.484,A -85,B 0,C 180,E1 -6992.165,E2 -6992.165} C_VEL
LIN {X 0,Y 481.666,Z 311.483,A -85,B 0,C 180,E1 -6994.967,E2 -6994.967} C_VEL
LIN {X 0,Y 481.641,Z 311.485,A -85,B 0,C 180,E1 -6997.704,E2 -6997.704} C_VEL
LIN {X 0,Y 481.694,Z 311.474,A -85,B 0,C 180,E1 -7000.393,E2 -7000.393} C_VEL
LIN {X 0,Y 481.665,Z 311.482,A -85,B 0,C 180,E1 -7003.033,E2 -7003.033} C_VEL
LIN {X 0,Y 481.678,Z 311.486,A -85,B 0,C 180,E1 -7005.638,E2 -7005.638} C_VEL
LIN {X 0,Y 481.742,Z 311.474,A -85,B 0,C 180,E1 -7008.215,E2 -7008.215} C_VEL
LIN {X 0,Y 481.721,Z 311.482,A -85,B 0,C 180,E1 -7011.611,E2 -7011.611} C_VEL
LIN {X 0,Y 481.786,Z 311.466,A -85,B 0,C 180,E1 -7014.139,E2 -7014.139} C_VEL
LIN {X 0,Y 481.898,Z 311.459,A -85,B 0,C 180,E1 -7017.492,E2 -7017.492} C_VEL
LIN {X 0,Y 481.9,Z 311.449,A -85,B 0,C 180,E1 -7020,E2 -7020} C_VEL
LIN {X 0,Y 481.906,Z 311.45,A -85,B 0,C 180,E1 -7022.508,E2 -7022.508} C_VEL
LIN {X 0,Y 481.767,Z 311.471,A -85,B 0,C 180,E1 -7025.861,E2 -7025.861} C_VEL
LIN {X 0,Y 481.726,Z 311.47,A -85,B 0,C 180,E1 -7028.389,E2 -7028.389} C_VEL
LIN {X 0,Y 481.742,Z 311.477,A -85,B 0,C 180,E1 -7031.785,E2 -7031.785} C_VEL
LIN {X 0,Y 481.729,Z 311.47,A -85,B 0,C 180,E1 -7035.225,E2 -7035.225} C_VEL
LIN {X 0,Y 481.697,Z 311.478,A -85,B 0,C 180,E1 -7038.722,E2 -7038.722} C_VEL
LIN {X 0,Y 481.637,Z 311.485,A -85,B 0,C 180,E1 -7041.395,E2 -7041.395} C_VEL
LIN {X 0,Y 481.64,Z 311.487,A -85,B 0,C 180,E1 -7044.115,E2 -7044.115} C_VEL
LIN {X 0,Y 481.646,Z 311.483,A -85,B 0,C 180,E1 -7047.118,E2 -7047.118} C_VEL
LIN {X 0,Y 481.65,Z 311.468,A -85,B 0,C 180,E1 -7049.743,E2 -7049.743} C_VEL
LIN {X 0,Y 481.646,Z 311.481,A -85,B 0,C 180,E1 -7052.676,E2 -7052.676} C_VEL
LIN {X 0,Y 481.624,Z 311.49,A -85,B 0,C 180,E1 -7055.711,E2 -7055.711} C_VEL
LIN {X 0,Y 481.628,Z 311.476,A -85,B 0,C 180,E1 -7058.864,E2 -7058.864} C_VEL
LIN {X 0,Y 481.616,Z 311.491,A -85,B 0,C 180,E1 -7061.909,E2 -7061.909} C_VEL
LIN {X 0,Y 481.649,Z 311.484,A -85,B 0,C 180,E1 -7064.459,E2 -7064.459} C_VEL
LIN {X 0,Y 481.611,Z 311.489,A -85,B 0,C 180,E1 -7067.836,E2 -7067.836} C_VEL
LIN {X 0,Y 481.645,Z 311.486,A -85,B 0,C 180,E1 -7070.657,E2 -7070.657} C_VEL
LIN {X 0,Y 481.615,Z 311.488,A -85,B 0,C 180,E1 -7073.379,E2 -7073.379} C_VEL
LIN {X 0,Y 481.669,Z 311.481,A -85,B 0,C 180,E1 -7076.327,E2 -7076.327} C_VEL
LIN {X 0,Y 481.626,Z 311.494,A -85,B 0,C 180,E1 -7079.423,E2 -7079.423} C_VEL
LIN {X 0,Y 481.645,Z 311.47,A -85,B 0,C 180,E1 -7082.165,E2 -7082.165} C_VEL
LIN {X 0,Y 481.665,Z 311.486,A -85,B 0,C 180,E1 -7084.968,E2 -7084.968} C_VEL
LIN {X 0,Y 481.635,Z 311.479,A -85,B 0,C 180,E1 -7087.94,E2 -7087.94} C_VEL
LIN {X 0,Y 480.965,Z 311.567,A -85,B 0,C 180,E1 -7088.638,E2 -7088.638} C_VEL
LIN {X 0,Y 478.133,Z 311.927,A -85,B 0,C 180,E1 -7089.772,E2 -7089.772} C_VEL
LIN {X 0,Y 475.74,Z 312.215,A -85,B 0,C 180,E1 -7090.686,E2 -7090.686} C_VEL
LIN {X 0,Y 474.71,Z 312.328,A -85,B 0,C 180,E1 -7091.392,E2 -7091.392} C_VEL
LIN {X 0,Y 474.625,Z 312.333,A -85,B 0,C 180,E1 -7091.631,E2 -7091.631} C_VEL
LIN {X 0,Y 474.664,Z 312.558,A -85,B 0,C 180,E1 -7093.551,E2 -7093.551} C_VEL
LIN {X 0,Y 474.921,Z 313.521,A -85,B 0,C 180,E1 -7093.686,E2 -7093.686} C_VEL
LIN {X 0,Y 478.307,Z 322.82,A -85,B 0,C 180,E1 -7093.969,E2 -7093.969} C_VEL
LIN {X 0,Y 477.924,Z 393.354,A -85,B 0,C 180,E1 -7095.061,E2 -7095.061} C_VEL
LIN {X 0,Y 477.796,Z 406.419,A -85,B 0,C 180,E1 -7095.438,E2 -7095.438} C_VEL
LIN {X 0,Y 477.615,Z 418.415,A -85,B 0,C 180,E1 -7095.949,E2 -7095.949} C_VEL
LIN {X 0,Y 477.347,Z 429.675,A -85,B 0,C 180,E1 -7096.591,E2 -7096.591} C_VEL
LIN {X 0,Y 476.866,Z 441.264,A -85,B 0,C 180,E1 -7097.445,E2 -7097.445} C_VEL
LIN {X 0,Y 476.435,Z 451.609,A -85,B 0,C 180,E1 -7098.406,E2 -7098.406} C_VEL
LIN {X 0,Y 476.086,Z 460.043,A -85,B 0,C 180,E1 -7099.367,E2 -7099.367} C_VEL
LIN {X 0,Y 475.67,Z 467.808,A -85,B 0,C 180,E1 -7100.432,E2 -7100.432} C_VEL
LIN {X 0,Y 475.327,Z 475.49,A -85,B 0,C 180,E1 -7101.733,E2 -7101.733} C_VEL
LIN {X 0,Y 475.065,Z 481.25,A -85,B 0,C 180,E1 -7102.946,E2 -7102.946} C_VEL
LIN {X 0,Y 474.922,Z 485.528,A -85,B 0,C 180,E1 -7104.054,E2 -7104.054} C_VEL
LIN {X 0,Y 474.647,Z 489.42,A -85,B 0,C 180,E1 -7105.329,E2 -7105.329} C_VEL
LIN {X 0,Y 474.462,Z 492.291,A -85,B 0,C 180,E1 -7106.603,E2 -7106.603} C_VEL
LIN {X 0,Y 474.498,Z 493.653,A -85,B 0,C 180,E1 -7107.453,E2 -7107.453} C_VEL
LIN {X 0,Y 474.378,Z 494.639,A -85,B 0,C 180,E1 -7108.302,E2 -7108.302} C_VEL
LIN {X 0,Y 474.452,Z 495.227,A -85,B 0,C 180,E1 -7109.151,E2 -7109.151} C_VEL
LIN {X 0,Y 474.436,Z 495.459,A -85,B 0,C 180,E1 -7110,E2 -7110} C_VEL
LIN {X 0,Y 474.452,Z 495.277,A -85,B 0,C 180,E1 -7110.849,E2 -7110.849} C_VEL
LIN {X 0,Y 474.378,Z 494.721,A -85,B 0,C 180,E1 -7111.698,E2 -7111.698} C_VEL
LIN {X 0,Y 474.497,Z 493.767,A -85,B 0,C 180,E1 -7112.547,E2 -7112.547} C_VEL
LIN {X 0,Y 474.457,Z 492.457,A -85,B 0,C 180,E1 -7113.397,E2 -7113.397} C_VEL
LIN {X 0,Y 474.642,Z 489.647,A -85,B 0,C 180,E1 -7114.671,E2 -7114.671} C_VEL
LIN {X 0,Y 474.913,Z 485.832,A -85,B 0,C 180,E1 -7115.946,E2 -7115.946} C_VEL
LIN {X 0,Y 475.034,Z 480.752,A -85,B 0,C 180,E1 -7117.268,E2 -7117.268} C_VEL
LIN {X 0,Y 475.447,Z 473.533,A -85,B 0,C 180,E1 -7118.715,E2 -7118.715} C_VEL
LIN {X 0,Y 475.881,Z 465.511,A -85,B 0,C 180,E1 -7119.993,E2 -7119.993} C_VEL
LIN {X 0,Y 476.242,Z 457.292,A -85,B 0,C 180,E1 -7121.06,E2 -7121.06} C_VEL
LIN {X 0,Y 476.618,Z 448.271,A -85,B 0,C 180,E1 -7122.021,E2 -7122.021} C_VEL
LIN {X 0,Y 477.103,Z 437.782,A -85,B 0,C 180,E1 -7122.922,E2 -7122.922} C_VEL
LIN {X 0,Y 477.394,Z 426.293,A -85,B 0,C 180,E1 -7123.711,E2 -7123.711} C_VEL
LIN {X 0,Y 477.67,Z 413.754,A -85,B 0,C 180,E1 -7124.365,E2 -7124.365} C_VEL
LIN {X 0,Y 477.843,Z 400.997,A -85,B 0,C 180,E1 -7124.833,E2 -7124.833} C_VEL
LIN {X 0,Y 477.868,Z 388.214,A -85,B 0,C 180,E1 -7125.132,E2 -7125.132} C_VEL
LIN {X 0,Y 478.205,Z 322.647,A -85,B 0,C 180,E1 -7126.13,E2 -7126.13} C_VEL
LIN {X 0,Y 474.783,Z 313.187,A -85,B 0,C 180,E1 -7126.434,E2 -7126.434} C_VEL
LIN {X 0,Y 474.623,Z 312.429,A -85,B 0,C 180,E1 -7126.6,E2 -7126.6} C_VEL
LIN {X 0,Y 474.612,Z 312.341,A -85,B 0,C 180,E1 -7129.012,E2 -7129.012} C_VEL
LIN {X 0,Y 474.585,Z 312.36,A -85,B 0,C 180,E1 -7131.729,E2 -7131.729} C_VEL
LIN {X 0,Y 474.619,Z 312.365,A -85,B 0,C 180,E1 -7134.495,E2 -7134.495} C_VEL
LIN {X 0,Y 474.592,Z 312.347,A -85,B 0,C 180,E1 -7137.326,E2 -7137.326} C_VEL
LIN {X 0,Y 474.579,Z 312.367,A -85,B 0,C 180,E1 -7140.231,E2 -7140.231} C_VEL
LIN {X 0,Y 474.606,Z 312.363,A -85,B 0,C 180,E1 -7143.222,E2 -7143.222} C_VEL
LIN {X 0,Y 474.577,Z 312.369,A -85,B 0,C 180,E1 -7146.324,E2 -7146.324} C_VEL
LIN {X 0,Y 474.597,Z 312.363,A -85,B 0,C 180,E1 -7149.643,E2 -7149.643} C_VEL
LIN {X 0,Y 474.571,Z 312.366,A -85,B 0,C 180,E1 -7152.229,E2 -7152.229} C_VEL
LIN {X 0,Y 474.608,Z 312.362,A -85,B 0,C 180,E1 -7155.298,E2 -7155.298} C_VEL
LIN {X 0,Y 474.586,Z 312.367,A -85,B 0,C 180,E1 -7158.211,E2 -7158.211} C_VEL
LIN {X 0,Y 474.613,Z 312.352,A -85,B 0,C 180,E1 -7160.451,E2 -7160.451} C_VEL
LIN {X 0,Y 474.576,Z 312.363,A -85,B 0,C 180,E1 -7163.675,E2 -7163.675} C_VEL
LIN {X 0,Y 474.608,Z 312.362,A -85,B 0,C 180,E1 -7166.777,E2 -7166.777} C_VEL
LIN {X 0,Y 474.578,Z 312.349,A -85,B 0,C 180,E1 -7169.768,E2 -7169.768} C_VEL
LIN {X 0,Y 474.595,Z 312.358,A -85,B 0,C 180,E1 -7172.684,E2 -7172.684} C_VEL
LIN {X 0,Y 474.617,Z 312.36,A -85,B 0,C 180,E1 -7175.505,E2 -7175.505} C_VEL
LIN {X 0,Y 474.643,Z 312.352,A -85,B 0,C 180,E1 -7179.184,E2 -7179.184} C_VEL
LIN {X 0,Y 474.629,Z 312.36,A -85,B 0,C 180,E1 -7181.883,E2 -7181.883} C_VEL
LIN {X 0,Y 474.688,Z 312.35,A -85,B 0,C 180,E1 -7184.544,E2 -7184.544} C_VEL
LIN {X 0,Y 474.695,Z 312.352,A -85,B 0,C 180,E1 -7188.037,E2 -7188.037} C_VEL
LIN {X 0,Y 474.658,Z 312.35,A -85,B 0,C 180,E1 -7191.485,E2 -7191.485} C_VEL
LIN {X 0,Y 474.719,Z 312.348,A -85,B 0,C 180,E1 -7194.052,E2 -7194.052} C_VEL
LIN {X 0,Y 474.872,Z 312.327,A -85,B 0,C 180,E1 -7197.455,E2 -7197.455} C_VEL
LIN {X 0,Y 474.868,Z 312.324,A -85,B 0,C 180,E1 -7200,E2 -7200} C_VEL
LIN {X 0,Y 474.862,Z 312.335,A -85,B 0,C 180,E1 -7202.545,E2 -7202.545} C_VEL
LIN {X 0,Y 474.748,Z 312.342,A -85,B 0,C 180,E1 -7205.948,E2 -7205.948} C_VEL
LIN {X 0,Y 474.692,Z 312.356,A -85,B 0,C 180,E1 -7208.514,E2 -7208.514} C_VEL
LIN {X 0,Y 474.684,Z 312.354,A -85,B 0,C 180,E1 -7211.963,E2 -7211.963} C_VEL
LIN {X 0,Y 474.691,Z 312.351,A -85,B 0,C 180,E1 -7215.456,E2 -7215.456} C_VEL
LIN {X 0,Y 474.653,Z 312.349,A -85,B 0,C 180,E1 -7219.011,E2 -7219.011} C_VEL
LIN {X 0,Y 474.58,Z 312.356,A -85,B 0,C 180,E1 -7221.729,E2 -7221.729} C_VEL
LIN {X 0,Y 474.619,Z 312.365,A -85,B 0,C 180,E1 -7224.495,E2 -7224.495} C_VEL
LIN {X 0,Y 474.631,Z 312.354,A -85,B 0,C 180,E1 -7227.324,E2 -7227.324} C_VEL
LIN {X 0,Y 474.596,Z 312.367,A -85,B 0,C 180,E1 -7230.231,E2 -7230.231} C_VEL
LIN {X 0,Y 474.609,Z 312.36,A -85,B 0,C 180,E1 -7233.223,E2 -7233.223} C_VEL
LIN {X 0,Y 474.564,Z 312.373,A -85,B 0,C 180,E1 -7236.326,E2 -7236.326} C_VEL
LIN {X 0,Y 474.595,Z 312.362,A -85,B 0,C 180,E1 -7239.644,E2 -7239.644} C_VEL
LIN {X 0,Y 474.57,Z 312.364,A -85,B 0,C 180,E1 -7242.939,E2 -7242.939} C_VEL
LIN {X 0,Y 474.576,Z 312.356,A -85,B 0,C 180,E1 -7245.892,E2 -7245.892} C_VEL
LIN {X 0,Y 474.596,Z 312.362,A -85,B 0,C 180,E1 -7249.046,E2 -7249.046} C_VEL
LIN {X 0,Y 474.587,Z 312.365,A -85,B 0,C 180,E1 -7251.708,E2 -7251.708} C_VEL
LIN {X 0,Y 474.608,Z 312.361,A -85,B 0,C 180,E1 -7254.725,E2 -7254.725} C_VEL
LIN {X 0,Y 474.624,Z 312.361,A -85,B 0,C 180,E1 -7257.787,E2 -7257.787} C_VEL
LIN {X 0,Y 474.644,Z 312.534,A -85,B 0,C 180,E1 -7260.049,E2 -7260.049} C_VEL
LIN {X 0,Y 477.756,Z 326.69,A -85,B 0,C 180,E1 -7262.18,E2 -7262.18} C_VEL
LIN {X 0,Y 478.047,Z 330.114,A -85,B 0,C 180,E1 -7262.657,E2 -7262.657} C_VEL
LIN {X 0,Y 477.195,Z 352.733,A -85,B 0,C 180,E1 -7265.646,E2 -7265.646} C_VEL
LIN {X 0,Y 476.319,Z 377.046,A -85,B 0,C 180,E1 -7268.808,E2 -7268.808} C_VEL
LIN {X 0,Y 475.581,Z 401.043,A -85,B 0,C 180,E1 -7271.921,E2 -7271.921} C_VEL
LIN {X 0,Y 475.295,Z 411.055,A -85,B 0,C 180,E1 -7273.198,E2 -7273.198} C_VEL
LIN {X 0,Y 477.807,Z 435.982,A -85,B 0,C 180,E1 -7273.681,E2 -7273.681} C_VEL
LIN {X 0,Y 477.273,Z 521.404,A -85,B 0,C 180,E1 -7274.985,E2 -7274.985} C_VEL
LIN {X 0,Y 476.811,Z 534.733,A -85,B 0,C 180,E1 -7275.352,E2 -7275.352} C_VEL
LIN {X 0,Y 476.366,Z 546.985,A -85,B 0,C 180,E1 -7275.857,E2 -7275.857} C_VEL
LIN {X 0,Y 475.801,Z 559.377,A -85,B 0,C 180,E1 -7276.548,E2 -7276.548} C_VEL
LIN {X 0,Y 475.33,Z 571.519,A -85,B 0,C 180,E1 -7277.436,E2 -7277.436} C_VEL
LIN {X 0,Y 474.908,Z 581.728,A -85,B 0,C 180,E1 -7278.368,E2 -7278.368} C_VEL
LIN {X 0,Y 474.609,Z 590.426,A -85,B 0,C 180,E1 -7279.333,E2 -7279.333} C_VEL
LIN {X 0,Y 474.304,Z 598.464,A -85,B 0,C 180,E1 -7280.404,E2 -7280.404} C_VEL
LIN {X 0,Y 474.155,Z 606.352,A -85,B 0,C 180,E1 -7281.691,E2 -7281.691} C_VEL
LIN {X 0,Y 474.028,Z 613.63,A -85,B 0,C 180,E1 -7283.188,E2 -7283.188} C_VEL
LIN {X 0,Y 474.018,Z 618.49,A -85,B 0,C 180,E1 -7284.47,E2 -7284.47} C_VEL
LIN {X 0,Y 474.089,Z 622.217,A -85,B 0,C 180,E1 -7285.749,E2 -7285.749} C_VEL
LIN {X 0,Y 474.072,Z 624.133,A -85,B 0,C 180,E1 -7286.6,E2 -7286.6} C_VEL
LIN {X 0,Y 474.05,Z 625.569,A -85,B 0,C 180,E1 -7287.451,E2 -7287.451} C_VEL
LIN {X 0,Y 474.155,Z 627.237,A -85,B 0,C 180,E1 -7289.151,E2 -7289.151} C_VEL
LIN {X 0,Y 474.145,Z 627.459,A -85,B 0,C 180,E1 -7290,E2 -7290} C_VEL
LIN {X 0,Y 474.155,Z 627.238,A -85,B 0,C 180,E1 -7290.849,E2 -7290.849} C_VEL
LIN {X 0,Y 474.05,Z 625.573,A -85,B 0,C 180,E1 -7292.549,E2 -7292.549} C_VEL
LIN {X 0,Y 474.072,Z 624.137,A -85,B 0,C 180,E1 -7293.4,E2 -7293.4} C_VEL
LIN {X 0,Y 474.053,Z 621.111,A -85,B 0,C 180,E1 -7294.677,E2 -7294.677} C_VEL
LIN {X 0,Y 474.072,Z 617.023,A -85,B 0,C 180,E1 -7295.956,E2 -7295.956} C_VEL
LIN {X 0,Y 474.095,Z 610.739,A -85,B 0,C 180,E1 -7297.453,E2 -7297.453} C_VEL
LIN {X 0,Y 474.167,Z 603.888,A -85,B 0,C 180,E1 -7298.738,E2 -7298.738} C_VEL
LIN {X 0,Y 474.399,Z 595.423,A -85,B 0,C 180,E1 -7300.024,E2 -7300.024} C_VEL
LIN {X 0,Y 474.722,Z 586.769,A -85,B 0,C 180,E1 -7301.096,E2 -7301.096} C_VEL
LIN {X 0,Y 475.194,Z 576.817,A -85,B 0,C 180,E1 -7302.103,E2 -7302.103} C_VEL
LIN {X 0,Y 475.59,Z 565.591,A -85,B 0,C 180,E1 -7303.024,E2 -7303.024} C_VEL
LIN {X 0,Y 476.036,Z 554.087,A -85,B 0,C 180,E1 -7303.772,E2 -7303.772} C_VEL
